Yaskawa INFORM job: DEMO_ROOF_UPPER_0625_3PAINT_21.JBI

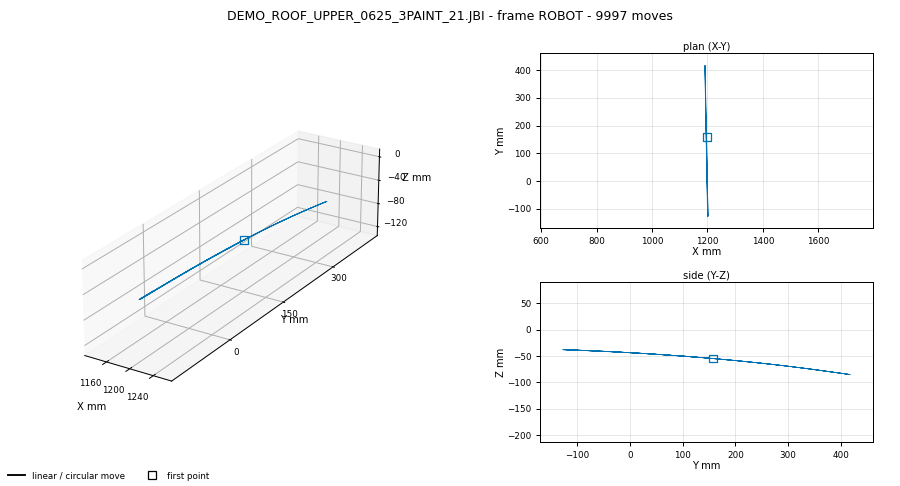
[picture p0: tool path of DEMO_ROOF_UPPER_0625_3PAINT_21.JBI in frame ROBOT, 9997 of 9997 moves have a stored position in this frame; points joined in program order, loops and branches not executed]
/JOB
//NAME DEMO_ROOF_UPPER_0625_3PAINT21
//POS
///NPOS 9997,0,0,0,0,0
///TOOL 0
///USER 0
///POSTYPE ROBOT
///RECTAN
///RCONF 1,0,0,0,0,0,0,0,0,0,0,0,0,0,0,0,0,0,0,0,0,0,0,0
C00000=1196.733,158.138,-54.632,-178.137,6.234,148.575
C00001=1196.739,157.889,-54.611,-178.140,6.232,148.575
C00002=1196.743,157.640,-54.589,-178.143,6.230,148.576
C00003=1196.748,157.391,-54.568,-178.145,6.229,148.576
C00004=1196.752,157.142,-54.547,-178.147,6.227,148.576
C00005=1196.757,156.894,-54.525,-178.150,6.226,148.577
C00006=1196.762,156.644,-54.504,-178.153,6.224,148.577
C00007=1196.766,156.395,-54.482,-178.156,6.222,148.578
C00008=1196.771,156.146,-54.460,-178.158,6.222,148.578
C00009=1196.776,155.896,-54.439,-178.161,6.220,148.579
C00010=1196.780,155.648,-54.418,-178.163,6.218,148.579
C00011=1196.785,155.399,-54.397,-178.166,6.216,148.579
C00012=1196.790,155.150,-54.375,-178.169,6.216,148.580
C00013=1196.795,154.900,-54.354,-178.171,6.214,148.580
C00014=1196.800,154.652,-54.332,-178.174,6.212,148.581
C00015=1196.804,154.403,-54.312,-178.177,6.210,148.581
C00016=1196.809,154.154,-54.290,-178.179,6.209,148.581
C00017=1196.813,153.904,-54.269,-178.182,6.208,148.582
C00018=1196.818,153.655,-54.247,-178.185,6.206,148.582
C00019=1196.823,153.406,-54.226,-178.187,6.204,148.583
C00020=1196.828,153.158,-54.205,-178.189,6.203,148.583
C00021=1196.832,152.908,-54.184,-178.192,6.201,148.584
C00022=1196.837,152.659,-54.162,-178.195,6.200,148.584
C00023=1196.841,152.410,-54.142,-178.198,6.198,148.585
C00024=1196.846,152.162,-54.120,-178.200,6.197,148.585
C00025=1196.852,151.912,-54.099,-178.203,6.196,148.585
C00026=1196.856,151.662,-54.078,-178.205,6.194,148.586
C00027=1196.860,151.414,-54.056,-178.208,6.192,148.586
C00028=1196.865,151.165,-54.036,-178.211,6.191,148.587
C00029=1196.871,150.916,-54.015,-178.213,6.190,148.587
C00030=1196.875,150.667,-53.993,-178.216,6.188,148.587
C00031=1196.880,150.418,-53.972,-178.219,6.186,148.588
C00032=1196.884,150.169,-53.950,-178.221,6.185,148.588
C00033=1196.889,149.920,-53.930,-178.224,6.184,148.589
C00034=1196.894,149.670,-53.909,-178.227,6.182,148.589
C00035=1196.899,149.421,-53.888,-178.229,6.180,148.590
C00036=1196.903,149.173,-53.867,-178.231,6.179,148.590
C00037=1196.908,148.924,-53.846,-178.235,6.178,148.591
C00038=1196.913,148.674,-53.825,-178.237,6.176,148.591
C00039=1196.917,148.425,-53.804,-178.239,6.175,148.591
C00040=1196.922,148.176,-53.783,-178.242,6.173,148.592
C00041=1196.927,147.927,-53.762,-178.245,6.171,148.592
C00042=1196.932,147.678,-53.741,-178.248,6.170,148.593
C00043=1196.937,147.429,-53.720,-178.250,6.169,148.593
C00044=1196.941,147.180,-53.699,-178.253,6.167,148.593
C00045=1196.946,146.930,-53.678,-178.255,6.165,148.594
C00046=1196.950,146.681,-53.658,-178.258,6.165,148.594
C00047=1196.955,146.432,-53.637,-178.261,6.163,148.595
C00048=1196.959,146.184,-53.616,-178.263,6.161,148.595
C00049=1196.965,145.934,-53.595,-178.266,6.159,148.596
C00050=1196.969,145.685,-53.574,-178.269,6.159,148.596
C00051=1196.974,145.436,-53.553,-178.271,6.157,148.597
C00052=1196.979,145.187,-53.533,-178.274,6.155,148.597
C00053=1196.984,144.938,-53.512,-178.276,6.154,148.597
C00054=1196.988,144.689,-53.492,-178.279,6.153,148.598
C00055=1196.993,144.440,-53.470,-178.282,6.151,148.598
C00056=1196.997,144.191,-53.449,-178.284,6.150,148.599
C00057=1197.002,143.942,-53.428,-178.287,6.148,148.599
C00058=1197.006,143.693,-53.408,-178.290,6.147,148.600
C00059=1197.012,143.443,-53.387,-178.293,6.145,148.600
C00060=1197.016,143.194,-53.366,-178.295,6.144,148.601
C00061=1197.021,142.945,-53.345,-178.297,6.142,148.601
C00062=1197.026,142.696,-53.325,-178.301,6.141,148.602
C00063=1197.031,142.447,-53.304,-178.303,6.140,148.602
C00064=1197.035,142.198,-53.284,-178.305,6.138,148.602
C00065=1197.041,141.949,-53.263,-178.308,6.137,148.603
C00066=1197.045,141.700,-53.242,-178.311,6.136,148.603
C00067=1197.049,141.451,-53.222,-178.313,6.134,148.604
C00068=1197.055,141.202,-53.201,-178.316,6.132,148.604
C00069=1197.059,140.953,-53.181,-178.318,6.131,148.604
C00070=1197.064,140.703,-53.160,-178.321,6.130,148.605
C00071=1197.069,140.454,-53.139,-178.324,6.128,148.605
C00072=1197.073,140.205,-53.119,-178.326,6.127,148.606
C00073=1197.078,139.956,-53.098,-178.329,6.126,148.606
C00074=1197.083,139.707,-53.078,-178.332,6.124,148.607
C00075=1197.087,139.458,-53.058,-178.334,6.123,148.607
C00076=1197.093,139.208,-53.037,-178.337,6.121,148.608
C00077=1197.097,138.959,-53.017,-178.340,6.120,148.608
C00078=1197.101,138.710,-52.996,-178.342,6.119,148.609
C00079=1197.107,138.461,-52.975,-178.345,6.117,148.609
C00080=1197.111,138.212,-52.955,-178.347,6.115,148.609
C00081=1197.115,137.963,-52.935,-178.350,6.115,148.610
C00082=1197.121,137.713,-52.914,-178.353,6.113,148.610
C00083=1197.125,137.465,-52.894,-178.355,6.111,148.611
C00084=1197.130,137.216,-52.874,-178.358,6.111,148.611
C00085=1197.135,136.966,-52.853,-178.361,6.109,148.612
C00086=1197.139,136.717,-52.832,-178.363,6.107,148.612
C00087=1197.144,136.468,-52.813,-178.365,6.106,148.613
C00088=1197.149,136.220,-52.793,-178.369,6.105,148.613
C00089=1197.154,135.970,-52.772,-178.371,6.103,148.614
C00090=1197.159,135.721,-52.751,-178.373,6.102,148.614
C00091=1197.164,135.472,-52.732,-178.377,6.101,148.615
C00092=1197.169,135.222,-52.711,-178.379,6.100,148.615
C00093=1197.173,134.974,-52.690,-178.381,6.098,148.615
C00094=1197.178,134.725,-52.670,-178.385,6.096,148.616
C00095=1197.182,134.475,-52.650,-178.387,6.096,148.616
C00096=1197.187,134.226,-52.630,-178.389,6.094,148.617
C00097=1197.192,133.977,-52.609,-178.393,6.092,148.617
C00098=1197.197,133.728,-52.590,-178.395,6.091,148.618
C00099=1197.202,133.479,-52.569,-178.397,6.090,148.618
C00100=1197.207,133.210,-52.548,-178.401,6.088,148.619
C00101=1197.211,132.941,-52.525,-178.403,6.087,148.619
C00102=1197.217,132.672,-52.504,-178.406,6.086,148.620
C00103=1197.222,132.404,-52.482,-178.409,6.084,148.620
C00104=1197.226,132.155,-52.462,-178.411,6.082,148.621
C00105=1197.232,131.906,-52.442,-178.414,6.082,148.621
C00106=1197.237,131.657,-52.422,-178.417,6.080,148.622
C00107=1197.241,131.408,-52.402,-178.419,6.078,148.622
C00108=1197.246,131.159,-52.381,-178.422,6.078,148.623
C00109=1197.251,130.909,-52.362,-178.425,6.076,148.623
C00110=1197.255,130.660,-52.341,-178.427,6.075,148.623
C00111=1197.260,130.411,-52.322,-178.430,6.073,148.624
C00112=1197.265,130.162,-52.302,-178.432,6.072,148.624
C00113=1197.270,129.913,-52.281,-178.435,6.071,148.625
C00114=1197.275,129.664,-52.261,-178.438,6.069,148.626
C00115=1197.279,129.414,-52.241,-178.440,6.068,148.626
C00116=1197.285,129.166,-52.221,-178.443,6.067,148.626
C00117=1197.289,128.916,-52.202,-178.446,6.065,148.627
C00118=1197.294,128.667,-52.181,-178.448,6.064,148.627
C00119=1197.298,128.418,-52.162,-178.451,6.062,148.628
C00120=1197.303,128.168,-52.142,-178.453,6.062,148.628
C00121=1197.308,127.920,-52.122,-178.456,6.060,148.629
C00122=1197.313,127.670,-52.102,-178.459,6.058,148.629
C00123=1197.317,127.421,-52.082,-178.461,6.058,148.630
C00124=1197.322,127.172,-52.062,-178.464,6.056,148.630
C00125=1197.327,126.924,-52.042,-178.466,6.055,148.631
C00126=1197.332,126.674,-52.023,-178.469,6.054,148.631
C00127=1197.337,126.424,-52.003,-178.471,6.053,148.632
C00128=1197.341,126.175,-51.983,-178.474,6.051,148.632
C00129=1197.346,125.927,-51.963,-178.477,6.049,148.633
C00130=1197.351,125.677,-51.944,-178.479,6.049,148.633
C00131=1197.356,125.428,-51.923,-178.482,6.047,148.634
C00132=1197.360,125.178,-51.904,-178.485,6.046,148.634
C00133=1197.366,124.930,-51.884,-178.487,6.044,148.634
C00134=1197.370,124.681,-51.864,-178.490,6.044,148.635
C00135=1197.375,124.431,-51.844,-178.493,6.042,148.635
C00136=1197.380,124.182,-51.825,-178.495,6.040,148.636
C00137=1197.385,123.933,-51.805,-178.498,6.040,148.636
C00138=1197.389,123.684,-51.785,-178.501,6.038,148.637
C00139=1197.394,123.434,-51.765,-178.503,6.037,148.638
C00140=1197.399,123.186,-51.747,-178.506,6.036,148.638
C00141=1197.403,122.936,-51.727,-178.508,6.035,148.638
C00142=1197.408,122.687,-51.707,-178.511,6.033,148.639
C00143=1197.413,122.438,-51.687,-178.514,6.031,148.639
C00144=1197.418,122.189,-51.668,-178.516,6.031,148.640
C00145=1197.423,121.939,-51.648,-178.519,6.029,148.640
C00146=1197.428,121.689,-51.628,-178.521,6.028,148.641
C00147=1197.433,121.441,-51.608,-178.524,6.027,148.641
C00148=1197.437,121.192,-51.589,-178.527,6.026,148.642
C00149=1197.441,120.942,-51.570,-178.529,6.024,148.642
C00150=1197.447,120.694,-51.550,-178.532,6.023,148.643
C00151=1197.451,120.444,-51.531,-178.535,6.022,148.643
C00152=1197.457,120.195,-51.511,-178.537,6.021,148.644
C00153=1197.461,119.946,-51.492,-178.540,6.019,148.644
C00154=1197.466,119.697,-51.471,-178.543,6.018,148.645
C00155=1197.471,119.448,-51.453,-178.545,6.017,148.645
C00156=1197.475,119.198,-51.433,-178.548,6.015,148.646
C00157=1197.480,118.949,-51.413,-178.550,6.014,148.646
C00158=1197.485,118.700,-51.394,-178.553,6.013,148.647
C00159=1197.489,118.451,-51.375,-178.555,6.012,148.647
C00160=1197.495,118.202,-51.356,-178.558,6.011,148.648
C00161=1197.499,117.952,-51.336,-178.561,6.010,148.648
C00162=1197.504,117.703,-51.316,-178.563,6.008,148.649
C00163=1197.510,117.454,-51.297,-178.566,6.007,148.649
C00164=1197.514,117.205,-51.278,-178.569,6.005,148.650
C00165=1197.519,116.956,-51.259,-178.571,6.005,148.650
C00166=1197.524,116.706,-51.239,-178.574,6.003,148.651
C00167=1197.528,116.457,-51.219,-178.577,6.003,148.651
C00168=1197.533,116.208,-51.201,-178.579,6.001,148.652
C00169=1197.538,115.959,-51.181,-178.581,6.000,148.652
C00170=1197.543,115.710,-51.162,-178.585,5.998,148.653
C00171=1197.547,115.460,-51.143,-178.587,5.998,148.653
C00172=1197.552,115.212,-51.123,-178.590,5.996,148.654
C00173=1197.557,114.962,-51.104,-178.592,5.995,148.654
C00174=1197.561,114.713,-51.085,-178.595,5.993,148.655
C00175=1197.567,114.463,-51.066,-178.597,5.993,148.655
C00176=1197.572,114.214,-51.046,-178.600,5.991,148.656
C00177=1197.577,113.965,-51.027,-178.603,5.990,148.656
C00178=1197.581,113.716,-51.008,-178.605,5.989,148.657
C00179=1197.586,113.467,-50.989,-178.608,5.988,148.657
C00180=1197.590,113.217,-50.970,-178.611,5.986,148.658
C00181=1197.596,112.969,-50.950,-178.613,5.985,148.658
C00182=1197.601,112.718,-50.931,-178.616,5.984,148.659
C00183=1197.605,112.470,-50.913,-178.618,5.983,148.659
C00184=1197.610,112.220,-50.893,-178.621,5.982,148.660
C00185=1197.615,111.971,-50.874,-178.623,5.981,148.660
C00186=1197.619,111.722,-50.855,-178.627,5.979,148.661
C00187=1197.625,111.473,-50.836,-178.629,5.978,148.661
C00188=1197.629,111.223,-50.817,-178.631,5.977,148.662
C00189=1197.634,110.974,-50.798,-178.634,5.976,148.662
C00190=1197.639,110.725,-50.778,-178.637,5.974,148.663
C00191=1197.644,110.476,-50.760,-178.639,5.974,148.663
C00192=1197.649,110.226,-50.741,-178.642,5.972,148.664
C00193=1197.653,109.978,-50.722,-178.645,5.971,148.664
C00194=1197.658,109.728,-50.702,-178.647,5.970,148.665
C00195=1197.663,109.479,-50.684,-178.650,5.969,148.665
C00196=1197.668,109.229,-50.665,-178.653,5.967,148.666
C00197=1197.672,108.981,-50.646,-178.655,5.966,148.666
C00198=1197.678,108.731,-50.627,-178.658,5.965,148.667
C00199=1197.682,108.482,-50.608,-178.660,5.964,148.667
C00200=1197.687,108.233,-50.589,-178.663,5.963,148.668
C00201=1197.692,107.983,-50.571,-178.665,5.962,148.668
C00202=1197.697,107.734,-50.551,-178.668,5.961,148.669
C00203=1197.701,107.485,-50.532,-178.671,5.959,148.669
C00204=1197.707,107.217,-50.512,-178.674,5.958,148.670
C00205=1197.712,106.949,-50.492,-178.676,5.957,148.670
C00206=1197.717,106.680,-50.472,-178.679,5.956,148.671
C00207=1197.722,106.412,-50.451,-178.682,5.955,148.672
C00208=1197.727,106.162,-50.432,-178.685,5.953,148.672
C00209=1197.732,105.913,-50.413,-178.687,5.953,148.673
C00210=1197.737,105.664,-50.395,-178.690,5.951,148.673
C00211=1197.742,105.414,-50.376,-178.692,5.950,148.674
C00212=1197.747,105.165,-50.358,-178.695,5.949,148.674
C00213=1197.752,104.916,-50.338,-178.698,5.948,148.675
C00214=1197.756,104.666,-50.320,-178.700,5.946,148.675
C00215=1197.761,104.418,-50.301,-178.703,5.946,148.676
C00216=1197.766,104.168,-50.283,-178.706,5.944,148.676
C00217=1197.770,103.919,-50.264,-178.708,5.943,148.677
C00218=1197.776,103.670,-50.245,-178.711,5.943,148.677
C00219=1197.780,103.420,-50.226,-178.713,5.941,148.678
C00220=1197.785,103.171,-50.208,-178.716,5.940,148.678
C00221=1197.790,102.922,-50.189,-178.719,5.938,148.679
C00222=1197.795,102.672,-50.171,-178.721,5.938,148.679
C00223=1197.800,102.423,-50.151,-178.724,5.936,148.680
C00224=1197.805,102.174,-50.133,-178.726,5.936,148.680
C00225=1197.809,101.924,-50.115,-178.729,5.935,148.681
C00226=1197.815,101.676,-50.096,-178.732,5.933,148.682
C00227=1197.820,101.426,-50.078,-178.734,5.932,148.682
C00228=1197.824,101.177,-50.059,-178.737,5.931,148.683
C00229=1197.829,100.928,-50.040,-178.739,5.930,148.683
C00230=1197.834,100.678,-50.022,-178.742,5.929,148.684
C00231=1197.838,100.429,-50.003,-178.745,5.928,148.684
C00232=1197.843,100.180,-49.985,-178.747,5.927,148.685
C00233=1197.849,99.931,-49.966,-178.750,5.925,148.685
C00234=1197.853,99.681,-49.947,-178.753,5.925,148.686
C00235=1197.858,99.432,-49.929,-178.755,5.923,148.686
C00236=1197.863,99.183,-49.911,-178.758,5.922,148.687
C00237=1197.868,98.934,-49.892,-178.760,5.922,148.687
C00238=1197.872,98.684,-49.874,-178.763,5.920,148.688
C00239=1197.877,98.435,-49.856,-178.765,5.919,148.688
C00240=1197.883,98.186,-49.837,-178.768,5.918,148.689
C00241=1197.887,97.937,-49.819,-178.771,5.917,148.689
C00242=1197.892,97.687,-49.800,-178.773,5.916,148.690
C00243=1197.897,97.438,-49.782,-178.776,5.915,148.690
C00244=1197.901,97.189,-49.764,-178.779,5.914,148.691
C00245=1197.906,96.939,-49.745,-178.781,5.912,148.691
C00246=1197.911,96.690,-49.727,-178.784,5.912,148.692
C00247=1197.916,96.441,-49.709,-178.786,5.911,148.693
C00248=1197.921,96.192,-49.691,-178.789,5.909,148.693
C00249=1197.926,95.942,-49.673,-178.791,5.908,148.694
C00250=1197.931,95.693,-49.653,-178.795,5.907,148.694
C00251=1197.935,95.444,-49.635,-178.797,5.906,148.695
C00252=1197.940,95.195,-49.617,-178.799,5.906,148.695
C00253=1197.945,94.945,-49.599,-178.802,5.904,148.696
C00254=1197.950,94.696,-49.581,-178.805,5.903,148.696
C00255=1197.955,94.446,-49.563,-178.807,5.903,148.697
C00256=1197.960,94.197,-49.544,-178.810,5.901,148.697
C00257=1197.965,93.948,-49.526,-178.813,5.900,148.698
C00258=1197.970,93.699,-49.507,-178.815,5.899,148.698
C00259=1197.974,93.449,-49.489,-178.818,5.898,148.699
C00260=1197.979,93.200,-49.471,-178.820,5.897,148.700
C00261=1197.984,92.951,-49.453,-178.823,5.896,148.700
C00262=1197.989,92.702,-49.435,-178.825,5.895,148.701
C00263=1197.994,92.453,-49.417,-178.828,5.894,148.701
C00264=1197.999,92.203,-49.399,-178.831,5.893,148.702
C00265=1198.003,91.953,-49.381,-178.833,5.892,148.702
C00266=1198.009,91.704,-49.362,-178.836,5.890,148.703
C00267=1198.013,91.455,-49.344,-178.839,5.890,148.703
C00268=1198.018,91.206,-49.326,-178.841,5.889,148.704
C00269=1198.023,90.956,-49.308,-178.844,5.887,148.704
C00270=1198.028,90.707,-49.290,-178.847,5.887,148.705
C00271=1198.033,90.458,-49.272,-178.849,5.886,148.706
C00272=1198.037,90.208,-49.254,-178.852,5.884,148.706
C00273=1198.042,89.959,-49.236,-178.854,5.884,148.707
C00274=1198.047,89.710,-49.218,-178.857,5.883,148.707
C00275=1198.052,89.461,-49.200,-178.859,5.881,148.708
C00276=1198.057,89.212,-49.182,-178.862,5.881,148.708
C00277=1198.062,88.962,-49.164,-178.864,5.880,148.709
C00278=1198.067,88.713,-49.146,-178.867,5.878,148.709
C00279=1198.072,88.463,-49.129,-178.870,5.878,148.710
C00280=1198.076,88.214,-49.111,-178.873,5.876,148.710
C00281=1198.081,87.964,-49.093,-178.875,5.876,148.711
C00282=1198.086,87.715,-49.075,-178.877,5.875,148.712
C00283=1198.091,87.466,-49.057,-178.881,5.873,148.712
C00284=1198.096,87.217,-49.039,-178.883,5.872,148.713
C00285=1198.101,86.968,-49.021,-178.885,5.872,148.713
C00286=1198.106,86.718,-49.003,-178.888,5.870,148.714
C00287=1198.111,86.469,-48.985,-178.891,5.869,148.714
C00288=1198.115,86.220,-48.968,-178.893,5.869,148.715
C00289=1198.120,85.971,-48.950,-178.896,5.867,148.715
C00290=1198.125,85.721,-48.932,-178.899,5.867,148.716
C00291=1198.130,85.472,-48.914,-178.901,5.866,148.716
C00292=1198.135,85.222,-48.897,-178.904,5.864,148.717
C00293=1198.140,84.973,-48.879,-178.906,5.863,148.718
C00294=1198.145,84.724,-48.861,-178.909,5.863,148.718
C00295=1198.149,84.474,-48.843,-178.912,5.861,148.719
C00296=1198.155,84.224,-48.825,-178.914,5.860,148.719
C00297=1198.159,83.975,-48.807,-178.917,5.860,148.720
C00298=1198.164,83.726,-48.790,-178.919,5.859,148.720
C00299=1198.169,83.477,-48.773,-178.922,5.858,148.721
C00300=1198.174,83.227,-48.755,-178.924,5.857,148.721
C00301=1198.179,82.978,-48.737,-178.927,5.856,148.722
C00302=1198.184,82.729,-48.719,-178.930,5.855,148.723
C00303=1198.189,82.479,-48.701,-178.932,5.854,148.723
C00304=1198.193,82.230,-48.684,-178.935,5.853,148.724
C00305=1198.198,81.981,-48.666,-178.938,5.852,148.724
C00306=1198.203,81.731,-48.649,-178.940,5.851,148.725
C00307=1198.208,81.482,-48.631,-178.942,5.850,148.725
C00308=1198.214,81.214,-48.613,-178.945,5.849,148.726
C00309=1198.219,80.946,-48.593,-178.948,5.848,148.727
C00310=1198.225,80.677,-48.574,-178.951,5.847,148.727
C00311=1198.229,80.409,-48.556,-178.954,5.846,148.728
C00312=1198.234,80.159,-48.538,-178.956,5.845,148.728
C00313=1198.239,79.910,-48.520,-178.959,5.844,148.729
C00314=1198.244,79.661,-48.502,-178.961,5.843,148.729
C00315=1198.249,79.411,-48.485,-178.964,5.842,148.730
C00316=1198.253,79.162,-48.468,-178.967,5.841,148.731
C00317=1198.258,78.912,-48.450,-178.969,5.840,148.731
C00318=1198.263,78.663,-48.432,-178.972,5.840,148.732
C00319=1198.268,78.415,-48.416,-178.974,5.839,148.732
C00320=1198.273,78.165,-48.398,-178.977,5.837,148.733
C00321=1198.279,77.916,-48.381,-178.980,5.837,148.734
C00322=1198.284,77.666,-48.363,-178.982,5.836,148.734
C00323=1198.288,77.417,-48.346,-178.985,5.834,148.735
C00324=1198.293,77.168,-48.328,-178.987,5.834,148.735
C00325=1198.298,76.918,-48.311,-178.990,5.833,148.736
C00326=1198.302,76.669,-48.294,-178.993,5.832,148.736
C00327=1198.308,76.419,-48.276,-178.995,5.831,148.737
C00328=1198.312,76.170,-48.258,-178.998,5.830,148.737
C00329=1198.317,75.921,-48.242,-179.000,5.829,148.738
C00330=1198.322,75.671,-48.224,-179.003,5.828,148.739
C00331=1198.328,75.422,-48.207,-179.006,5.827,148.739
C00332=1198.332,75.173,-48.190,-179.008,5.826,148.740
C00333=1198.337,74.924,-48.172,-179.011,5.826,148.740
C00334=1198.342,74.674,-48.155,-179.014,5.824,148.741
C00335=1198.347,74.424,-48.138,-179.016,5.824,148.741
C00336=1198.352,74.175,-48.120,-179.019,5.823,148.742
C00337=1198.357,73.925,-48.103,-179.021,5.822,148.742
C00338=1198.361,73.677,-48.086,-179.024,5.821,148.743
C00339=1198.367,73.427,-48.069,-179.027,5.820,148.744
C00340=1198.371,73.178,-48.052,-179.029,5.819,148.744
C00341=1198.376,72.929,-48.034,-179.032,5.819,148.745
C00342=1198.381,72.679,-48.017,-179.034,5.817,148.745
C00343=1198.386,72.429,-48.000,-179.037,5.816,148.746
C00344=1198.391,72.180,-47.983,-179.039,5.816,148.747
C00345=1198.396,71.932,-47.966,-179.042,5.815,148.747
C00346=1198.401,71.682,-47.949,-179.045,5.814,148.748
C00347=1198.406,71.432,-47.932,-179.047,5.813,148.748
C00348=1198.411,71.183,-47.914,-179.050,5.812,148.749
C00349=1198.415,70.934,-47.897,-179.052,5.812,148.749
C00350=1198.420,70.684,-47.880,-179.055,5.810,148.750
C00351=1198.425,70.435,-47.864,-179.058,5.809,148.751
C00352=1198.430,70.186,-47.846,-179.060,5.809,148.751
C00353=1198.435,69.936,-47.828,-179.062,5.808,148.752
C00354=1198.440,69.687,-47.812,-179.066,5.807,148.752
C00355=1198.446,69.437,-47.795,-179.068,5.806,148.753
C00356=1198.450,69.188,-47.778,-179.070,5.805,148.753
C00357=1198.454,68.939,-47.761,-179.073,5.805,148.754
C00358=1198.460,68.689,-47.744,-179.076,5.803,148.755
C00359=1198.464,68.440,-47.727,-179.078,5.802,148.755
C00360=1198.470,68.191,-47.710,-179.081,5.802,148.756
C00361=1198.474,67.941,-47.693,-179.083,5.801,148.756
C00362=1198.480,67.691,-47.676,-179.086,5.800,148.757
C00363=1198.484,67.442,-47.659,-179.089,5.799,148.758
C00364=1198.490,67.194,-47.642,-179.091,5.798,148.758
C00365=1198.494,66.944,-47.625,-179.094,5.797,148.759
C00366=1198.499,66.694,-47.608,-179.096,5.797,148.759
C00367=1198.504,66.445,-47.591,-179.099,5.795,148.760
C00368=1198.509,66.196,-47.575,-179.102,5.795,148.760
C00369=1198.514,65.946,-47.558,-179.104,5.794,148.761
C00370=1198.519,65.697,-47.541,-179.106,5.793,148.761
C00371=1198.524,65.447,-47.524,-179.109,5.793,148.762
C00372=1198.529,65.198,-47.507,-179.112,5.791,148.763
C00373=1198.533,64.949,-47.491,-179.114,5.790,148.763
C00374=1198.539,64.699,-47.473,-179.117,5.790,148.764
C00375=1198.543,64.449,-47.457,-179.120,5.789,148.765
C00376=1198.548,64.201,-47.441,-179.122,5.788,148.765
C00377=1198.553,63.951,-47.423,-179.125,5.787,148.766
C00378=1198.558,63.701,-47.407,-179.128,5.786,148.766
C00379=1198.564,63.452,-47.390,-179.130,5.786,148.767
C00380=1198.568,63.203,-47.373,-179.132,5.785,148.767
C00381=1198.573,62.953,-47.356,-179.135,5.784,148.768
C00382=1198.578,62.704,-47.339,-179.138,5.783,148.768
C00383=1198.583,62.455,-47.323,-179.140,5.782,148.769
C00384=1198.587,62.205,-47.306,-179.143,5.781,148.770
C00385=1198.593,61.956,-47.289,-179.145,5.781,148.770
C00386=1198.598,61.707,-47.273,-179.148,5.780,148.771
C00387=1198.602,61.457,-47.256,-179.151,5.778,148.771
C00388=1198.607,61.208,-47.240,-179.153,5.778,148.772
C00389=1198.613,60.958,-47.223,-179.156,5.777,148.773
C00390=1198.617,60.708,-47.206,-179.158,5.776,148.773
C00391=1198.622,60.460,-47.190,-179.161,5.776,148.774
C00392=1198.628,60.210,-47.173,-179.164,5.775,148.774
C00393=1198.632,59.960,-47.156,-179.166,5.774,148.775
C00394=1198.637,59.712,-47.140,-179.169,5.773,148.776
C00395=1198.642,59.462,-47.123,-179.171,5.773,148.776
C00396=1198.648,59.212,-47.107,-179.174,5.772,148.777
C00397=1198.652,58.963,-47.090,-179.176,5.771,148.777
C00398=1198.657,58.713,-47.074,-179.179,5.770,148.778
C00399=1198.662,58.465,-47.057,-179.182,5.769,148.779
C00400=1198.666,58.215,-47.041,-179.184,5.768,148.779
C00401=1198.672,57.965,-47.024,-179.187,5.768,148.780
C00402=1198.677,57.716,-47.008,-179.189,5.767,148.780
C00403=1198.681,57.466,-46.991,-179.191,5.766,148.781
C00404=1198.686,57.218,-46.975,-179.195,5.765,148.781
C00405=1198.692,56.968,-46.958,-179.197,5.764,148.782
C00406=1198.697,56.718,-46.942,-179.199,5.764,148.783
C00407=1198.702,56.469,-46.925,-179.202,5.763,148.783
C00408=1198.706,56.220,-46.909,-179.205,5.763,148.784
C00409=1198.711,55.970,-46.893,-179.207,5.762,148.784
C00410=1198.716,55.721,-46.876,-179.210,5.760,148.785
C00411=1198.722,55.472,-46.859,-179.213,5.760,148.786
C00412=1198.727,55.202,-46.842,-179.215,5.759,148.786
C00413=1198.732,54.934,-46.824,-179.218,5.759,148.787
C00414=1198.737,54.666,-46.807,-179.221,5.757,148.787
C00415=1198.742,54.397,-46.789,-179.223,5.756,148.788
C00416=1198.747,54.148,-46.774,-179.226,5.756,148.789
C00417=1198.753,53.898,-46.756,-179.229,5.755,148.789
C00418=1198.758,53.649,-46.740,-179.231,5.754,148.790
C00419=1198.763,53.399,-46.724,-179.234,5.753,148.791
C00420=1198.768,53.151,-46.708,-179.237,5.753,148.791
C00421=1198.772,52.900,-46.692,-179.239,5.752,148.792
C00422=1198.778,52.652,-46.676,-179.241,5.751,148.792
C00423=1198.782,52.402,-46.659,-179.244,5.751,148.793
C00424=1198.787,52.153,-46.643,-179.247,5.750,148.794
C00425=1198.792,51.903,-46.627,-179.249,5.749,148.794
C00426=1198.797,51.654,-46.611,-179.252,5.748,148.795
C00427=1198.802,51.404,-46.594,-179.255,5.747,148.795
C00428=1198.807,51.155,-46.579,-179.257,5.746,148.796
C00429=1198.812,50.906,-46.562,-179.259,5.746,148.797
C00430=1198.817,50.657,-46.546,-179.262,5.745,148.797
C00431=1198.821,50.407,-46.530,-179.265,5.745,148.798
C00432=1198.827,50.158,-46.514,-179.267,5.744,148.798
C00433=1198.831,49.908,-46.498,-179.270,5.743,148.799
C00434=1198.837,49.659,-46.481,-179.273,5.742,148.800
C00435=1198.842,49.409,-46.465,-179.275,5.741,148.800
C00436=1198.846,49.160,-46.449,-179.278,5.741,148.801
C00437=1198.851,48.910,-46.433,-179.280,5.740,148.801
C00438=1198.856,48.661,-46.418,-179.283,5.739,148.802
C00439=1198.861,48.411,-46.401,-179.285,5.739,148.803
C00440=1198.866,48.162,-46.385,-179.288,5.738,148.803
C00441=1198.871,47.912,-46.369,-179.290,5.738,148.804
C00442=1198.876,47.663,-46.353,-179.293,5.736,148.804
C00443=1198.881,47.414,-46.337,-179.296,5.735,148.805
C00444=1198.886,47.164,-46.321,-179.298,5.735,148.806
C00445=1198.891,46.915,-46.305,-179.301,5.734,148.806
C00446=1198.896,46.665,-46.288,-179.303,5.733,148.807
C00447=1198.901,46.416,-46.273,-179.306,5.733,148.807
C00448=1198.906,46.166,-46.256,-179.308,5.732,148.808
C00449=1198.911,45.917,-46.241,-179.310,5.731,148.809
C00450=1198.917,45.667,-46.225,-179.313,5.731,148.809
C00451=1198.921,45.418,-46.208,-179.316,5.730,148.810
C00452=1198.926,45.168,-46.193,-179.319,5.729,148.811
C00453=1198.930,44.919,-46.177,-179.321,5.728,148.811
C00454=1198.936,44.670,-46.161,-179.324,5.728,148.812
C00455=1198.941,44.421,-46.146,-179.326,5.727,148.812
C00456=1198.946,44.170,-46.130,-179.329,5.726,148.813
C00457=1198.951,43.921,-46.114,-179.331,5.726,148.813
C00458=1198.956,43.672,-46.098,-179.334,5.725,148.814
C00459=1198.961,43.422,-46.082,-179.336,5.725,148.815
C00460=1198.966,43.173,-46.066,-179.339,5.724,148.815
C00461=1198.970,42.924,-46.050,-179.341,5.723,148.816
C00462=1198.975,42.674,-46.034,-179.344,5.722,148.817
C00463=1198.981,42.425,-46.019,-179.347,5.721,148.817
C00464=1198.986,42.175,-46.003,-179.349,5.720,148.818
C00465=1198.991,41.925,-45.987,-179.352,5.720,148.818
C00466=1198.996,41.676,-45.971,-179.355,5.719,148.819
C00467=1199.000,41.427,-45.956,-179.357,5.718,148.820
C00468=1199.006,41.177,-45.940,-179.359,5.718,148.820
C00469=1199.011,40.928,-45.925,-179.362,5.717,148.821
C00470=1199.016,40.678,-45.909,-179.365,5.717,148.822
C00471=1199.021,40.429,-45.892,-179.367,5.716,148.822
C00472=1199.025,40.180,-45.877,-179.369,5.715,148.823
C00473=1199.030,39.930,-45.861,-179.372,5.715,148.823
C00474=1199.036,39.680,-45.846,-179.375,5.714,148.824
C00475=1199.041,39.431,-45.830,-179.377,5.713,148.824
C00476=1199.046,39.182,-45.815,-179.380,5.712,148.825
C00477=1199.050,38.932,-45.799,-179.383,5.712,148.826
C00478=1199.056,38.683,-45.783,-179.385,5.711,148.826
C00479=1199.061,38.434,-45.767,-179.387,5.710,148.827
C00480=1199.065,38.184,-45.752,-179.390,5.710,148.828
C00481=1199.070,37.934,-45.736,-179.393,5.709,148.828
C00482=1199.076,37.685,-45.721,-179.395,5.709,148.829
C00483=1199.081,37.436,-45.705,-179.398,5.708,148.829
C00484=1199.085,37.186,-45.690,-179.400,5.707,148.830
C00485=1199.091,36.936,-45.674,-179.403,5.707,148.831
C00486=1199.096,36.687,-45.659,-179.405,5.706,148.831
C00487=1199.101,36.438,-45.644,-179.408,5.705,148.832
C00488=1199.105,36.188,-45.628,-179.410,5.705,148.833
C00489=1199.111,35.938,-45.612,-179.413,5.704,148.833
C00490=1199.115,35.689,-45.597,-179.416,5.704,148.834
C00491=1199.121,35.440,-45.582,-179.418,5.702,148.834
C00492=1199.126,35.190,-45.566,-179.421,5.702,148.835
C00493=1199.130,34.941,-45.551,-179.424,5.701,148.836
C00494=1199.136,34.691,-45.535,-179.426,5.700,148.836
C00495=1199.141,34.442,-45.519,-179.428,5.700,148.837
C00496=1199.145,34.192,-45.504,-179.431,5.699,148.837
C00497=1199.150,33.943,-45.488,-179.434,5.699,148.838
C00498=1199.156,33.693,-45.473,-179.436,5.698,148.839
C00499=1199.160,33.444,-45.458,-179.438,5.697,148.839
C00500=1199.165,33.194,-45.442,-179.441,5.697,148.840
C00501=1199.170,32.945,-45.427,-179.444,5.696,148.841
C00502=1199.175,32.696,-45.411,-179.446,5.696,148.841
C00503=1199.181,32.446,-45.396,-179.449,5.695,148.842
C00504=1199.186,32.196,-45.381,-179.451,5.694,148.842
C00505=1199.190,31.946,-45.366,-179.454,5.694,148.843
C00506=1199.195,31.697,-45.351,-179.456,5.693,148.844
C00507=1199.200,31.448,-45.335,-179.459,5.692,148.844
C00508=1199.205,31.199,-45.320,-179.461,5.692,148.845
C00509=1199.211,30.949,-45.304,-179.464,5.691,148.846
C00510=1199.216,30.700,-45.289,-179.467,5.691,148.846
C00511=1199.220,30.450,-45.274,-179.469,5.690,148.847
C00512=1199.226,30.200,-45.259,-179.471,5.689,148.847
C00513=1199.230,29.951,-45.244,-179.474,5.689,148.848
C00514=1199.236,29.702,-45.228,-179.477,5.688,148.849
C00515=1199.240,29.453,-45.213,-179.479,5.688,148.849
C00516=1199.246,29.183,-45.197,-179.483,5.686,148.850
C00517=1199.251,28.915,-45.181,-179.485,5.686,148.851
C00518=1199.257,28.646,-45.164,-179.488,5.685,148.851
C00519=1199.263,28.377,-45.148,-179.490,5.685,148.852
C00520=1199.267,28.128,-45.133,-179.493,5.684,148.853
C00521=1199.272,27.878,-45.117,-179.495,5.684,148.853
C00522=1199.277,27.628,-45.102,-179.498,5.683,148.854
C00523=1199.282,27.379,-45.087,-179.501,5.682,148.855
C00524=1199.287,27.130,-45.072,-179.503,5.682,148.855
C00525=1199.292,26.881,-45.057,-179.505,5.681,148.856
C00526=1199.298,26.631,-45.042,-179.508,5.681,148.856
C00527=1199.302,26.382,-45.027,-179.511,5.680,148.857
C00528=1199.308,26.132,-45.011,-179.513,5.679,148.858
C00529=1199.312,25.882,-44.997,-179.515,5.679,148.858
C00530=1199.317,25.632,-44.981,-179.518,5.678,148.859
C00531=1199.322,25.383,-44.966,-179.521,5.678,148.860
C00532=1199.327,25.133,-44.952,-179.523,5.677,148.860
C00533=1199.332,24.884,-44.936,-179.526,5.676,148.861
C00534=1199.337,24.635,-44.921,-179.528,5.676,148.861
C00535=1199.343,24.385,-44.906,-179.531,5.675,148.862
C00536=1199.347,24.136,-44.891,-179.533,5.675,148.863
C00537=1199.352,23.886,-44.877,-179.536,5.674,148.863
C00538=1199.358,23.637,-44.862,-179.538,5.673,148.864
C00539=1199.362,23.388,-44.847,-179.541,5.673,148.865
C00540=1199.368,23.138,-44.832,-179.544,5.672,148.865
C00541=1199.373,22.889,-44.817,-179.546,5.672,148.866
C00542=1199.378,22.639,-44.802,-179.548,5.671,148.866
C00543=1199.383,22.389,-44.787,-179.551,5.670,148.867
C00544=1199.388,22.140,-44.773,-179.554,5.670,148.868
C00545=1199.393,21.891,-44.758,-179.556,5.669,148.868
C00546=1199.397,21.641,-44.742,-179.559,5.669,148.869
C00547=1199.402,21.391,-44.727,-179.561,5.668,148.870
C00548=1199.407,21.142,-44.712,-179.564,5.667,148.870
C00549=1199.413,20.892,-44.698,-179.566,5.667,148.871
C00550=1199.417,20.643,-44.683,-179.569,5.666,148.872
C00551=1199.422,20.393,-44.668,-179.571,5.666,148.872
C00552=1199.428,20.144,-44.653,-179.574,5.665,148.873
C00553=1199.433,19.894,-44.638,-179.577,5.665,148.873
C00554=1199.438,19.644,-44.624,-179.579,5.664,148.874
C00555=1199.443,19.395,-44.609,-179.582,5.664,148.875
C00556=1199.448,19.145,-44.594,-179.584,5.663,148.875
C00557=1199.453,18.896,-44.579,-179.587,5.662,148.876
C00558=1199.457,18.646,-44.565,-179.589,5.662,148.877
C00559=1199.463,18.397,-44.549,-179.592,5.661,148.877
C00560=1199.468,18.147,-44.535,-179.595,5.661,148.878
C00561=1199.473,17.898,-44.521,-179.597,5.660,148.878
C00562=1199.478,17.649,-44.506,-179.599,5.660,148.879
C00563=1199.484,17.399,-44.491,-179.601,5.660,148.880
C00564=1199.488,17.150,-44.476,-179.604,5.659,148.880
C00565=1199.493,16.900,-44.462,-179.607,5.659,148.881
C00566=1199.498,16.650,-44.448,-179.609,5.658,148.882
C00567=1199.503,16.401,-44.433,-179.612,5.657,148.882
C00568=1199.509,16.151,-44.418,-179.614,5.657,148.883
C00569=1199.514,15.902,-44.404,-179.617,5.656,148.884
C00570=1199.518,15.653,-44.389,-179.620,5.656,148.884
C00571=1199.523,15.403,-44.374,-179.622,5.655,148.885
C00572=1199.528,15.153,-44.360,-179.624,5.654,148.885
C00573=1199.534,14.904,-44.344,-179.627,5.654,148.886
C00574=1199.538,14.654,-44.330,-179.630,5.653,148.887
C00575=1199.543,14.404,-44.316,-179.632,5.653,148.888
C00576=1199.548,14.155,-44.301,-179.634,5.652,148.888
C00577=1199.553,13.905,-44.287,-179.637,5.651,148.889
C00578=1199.559,13.656,-44.273,-179.640,5.651,148.889
C00579=1199.564,13.406,-44.258,-179.642,5.650,148.890
C00580=1199.569,13.157,-44.243,-179.645,5.650,148.891
C00581=1199.574,12.908,-44.229,-179.647,5.650,148.891
C00582=1199.579,12.658,-44.214,-179.649,5.649,148.892
C00583=1199.584,12.408,-44.200,-179.652,5.649,148.893
C00584=1199.588,12.159,-44.185,-179.655,5.648,148.893
C00585=1199.593,11.909,-44.171,-179.657,5.648,148.894
C00586=1199.598,11.660,-44.157,-179.659,5.647,148.894
C00587=1199.605,11.410,-44.142,-179.662,5.646,148.895
C00588=1199.610,11.161,-44.128,-179.665,5.646,148.896
C00589=1199.614,10.912,-44.113,-179.667,5.645,148.896
C00590=1199.619,10.662,-44.098,-179.670,5.645,148.897
C00591=1199.624,10.412,-44.084,-179.672,5.644,148.898
C00592=1199.629,10.162,-44.070,-179.675,5.644,148.898
C00593=1199.634,9.913,-44.056,-179.677,5.643,148.899
C00594=1199.640,9.664,-44.042,-179.680,5.643,148.900
C00595=1199.645,9.414,-44.027,-179.683,5.642,148.900
C00596=1199.649,9.165,-44.012,-179.684,5.642,148.901
C00597=1199.654,8.915,-43.998,-179.687,5.642,148.901
C00598=1199.659,8.666,-43.984,-179.690,5.641,148.902
C00599=1199.664,8.416,-43.970,-179.692,5.641,148.903
C00600=1199.670,8.167,-43.956,-179.695,5.640,148.903
C00601=1199.675,7.917,-43.941,-179.697,5.639,148.904
C00602=1199.680,7.667,-43.927,-179.700,5.639,148.905
C00603=1199.685,7.418,-43.913,-179.702,5.638,148.905
C00604=1199.689,7.168,-43.899,-179.705,5.638,148.906
C00605=1199.695,6.919,-43.885,-179.708,5.637,148.907
C00606=1199.700,6.669,-43.870,-179.710,5.637,148.907
C00607=1199.705,6.420,-43.856,-179.712,5.637,148.908
C00608=1199.710,6.170,-43.842,-179.715,5.636,148.909
C00609=1199.715,5.920,-43.828,-179.717,5.636,148.909
C00610=1199.720,5.671,-43.814,-179.720,5.635,148.910
C00611=1199.725,5.421,-43.799,-179.723,5.635,148.911
C00612=1199.730,5.172,-43.785,-179.725,5.634,148.911
C00613=1199.735,4.922,-43.771,-179.727,5.633,148.912
C00614=1199.740,4.672,-43.757,-179.730,5.633,148.912
C00615=1199.746,4.423,-43.743,-179.733,5.632,148.913
C00616=1199.751,4.174,-43.728,-179.735,5.632,148.914
C00617=1199.756,3.924,-43.714,-179.737,5.632,148.914
C00618=1199.761,3.674,-43.700,-179.740,5.631,148.915
C00619=1199.766,3.425,-43.686,-179.742,5.631,148.916
C00620=1199.772,3.156,-43.671,-179.745,5.630,148.916
C00621=1199.777,2.887,-43.655,-179.747,5.630,148.917
C00622=1199.782,2.617,-43.640,-179.750,5.629,148.918
C00623=1199.788,2.348,-43.625,-179.753,5.629,148.918
C00624=1199.793,2.099,-43.611,-179.755,5.628,148.919
C00625=1199.798,1.849,-43.597,-179.758,5.628,148.920
C00626=1199.802,1.600,-43.583,-179.761,5.627,148.920
C00627=1199.807,1.350,-43.569,-179.763,5.627,148.921
C00628=1199.813,1.101,-43.555,-179.766,5.626,148.922
C00629=1199.818,0.852,-43.541,-179.768,5.625,148.922
C00630=1199.823,0.601,-43.527,-179.771,5.625,148.923
C00631=1199.829,0.352,-43.513,-179.773,5.625,148.924
C00632=1199.834,0.102,-43.499,-179.776,5.625,148.924
C00633=1199.838,-0.147,-43.485,-179.778,5.624,148.925
C00634=1199.843,-0.396,-43.472,-179.780,5.623,148.925
C00635=1199.848,-0.646,-43.457,-179.783,5.623,148.926
C00636=1199.854,-0.896,-43.444,-179.786,5.622,148.927
C00637=1199.859,-1.145,-43.430,-179.788,5.622,148.928
C00638=1199.863,-1.394,-43.416,-179.791,5.621,148.928
C00639=1199.868,-1.644,-43.402,-179.793,5.621,148.929
C00640=1199.874,-1.894,-43.388,-179.795,5.621,148.929
C00641=1199.879,-2.143,-43.374,-179.798,5.620,148.930
C00642=1199.884,-2.393,-43.360,-179.801,5.620,148.931
C00643=1199.888,-2.643,-43.346,-179.803,5.619,148.931
C00644=1199.894,-2.892,-43.333,-179.806,5.619,148.932
C00645=1199.899,-3.142,-43.319,-179.808,5.618,148.933
C00646=1199.905,-3.391,-43.305,-179.811,5.618,148.933
C00647=1199.909,-3.640,-43.291,-179.813,5.618,148.934
C00648=1199.914,-3.891,-43.278,-179.815,5.617,148.935
C00649=1199.920,-4.140,-43.264,-179.818,5.617,148.935
C00650=1199.925,-4.389,-43.250,-179.821,5.616,148.936
C00651=1199.929,-4.639,-43.237,-179.823,5.616,148.937
C00652=1199.935,-4.888,-43.223,-179.826,5.615,148.937
C00653=1199.940,-5.138,-43.208,-179.828,5.615,148.938
C00654=1199.945,-5.388,-43.195,-179.830,5.615,148.939
C00655=1199.950,-5.637,-43.182,-179.833,5.614,148.939
C00656=1199.955,-5.887,-43.167,-179.836,5.614,148.940
C00657=1199.961,-6.136,-43.154,-179.838,5.613,148.940
C00658=1199.965,-6.386,-43.140,-179.840,5.613,148.941
C00659=1199.970,-6.636,-43.127,-179.843,5.612,148.942
C00660=1199.976,-6.885,-43.113,-179.846,5.612,148.943
C00661=1199.980,-7.135,-43.099,-179.848,5.612,148.943
C00662=1199.986,-7.384,-43.086,-179.850,5.611,148.944
C00663=1199.991,-7.634,-43.072,-179.853,5.611,148.944
C00664=1199.995,-7.884,-43.059,-179.855,5.610,148.945
C00665=1200.001,-8.133,-43.045,-179.858,5.610,148.946
C00666=1200.006,-8.383,-43.031,-179.861,5.609,148.946
C00667=1200.011,-8.632,-43.018,-179.863,5.609,148.947
C00668=1200.016,-8.882,-43.004,-179.865,5.609,148.948
C00669=1200.022,-9.131,-42.991,-179.868,5.608,148.948
C00670=1200.026,-9.381,-42.977,-179.870,5.608,148.949
C00671=1200.031,-9.631,-42.963,-179.873,5.607,148.950
C00672=1200.036,-9.880,-42.950,-179.875,5.607,148.950
C00673=1200.041,-10.130,-42.936,-179.878,5.607,148.951
C00674=1200.047,-10.379,-42.923,-179.880,5.607,148.952
C00675=1200.051,-10.629,-42.910,-179.882,5.606,148.952
C00676=1200.057,-10.878,-42.896,-179.885,5.605,148.953
C00677=1200.061,-11.128,-42.883,-179.888,5.605,148.954
C00678=1200.067,-11.377,-42.869,-179.890,5.604,148.954
C00679=1200.072,-11.627,-42.855,-179.892,5.605,148.955
C00680=1200.077,-11.877,-42.843,-179.895,5.604,148.956
C00681=1200.082,-12.126,-42.828,-179.897,5.603,148.956
C00682=1200.087,-12.376,-42.816,-179.900,5.603,148.957
C00683=1200.092,-12.626,-42.801,-179.903,5.602,148.957
C00684=1200.097,-12.875,-42.789,-179.905,5.602,148.958
C00685=1200.102,-13.125,-42.775,-179.907,5.602,148.959
C00686=1200.107,-13.374,-42.762,-179.910,5.602,148.960
C00687=1200.113,-13.624,-42.748,-179.912,5.601,148.960
C00688=1200.118,-13.873,-42.734,-179.915,5.600,148.961
C00689=1200.123,-14.123,-42.722,-179.917,5.600,148.961
C00690=1200.129,-14.373,-42.708,-179.920,5.600,148.962
C00691=1200.133,-14.622,-42.695,-179.922,5.600,148.963
C00692=1200.139,-14.872,-42.681,-179.925,5.599,148.964
C00693=1200.143,-15.121,-42.668,-179.927,5.598,148.964
C00694=1200.149,-15.371,-42.655,-179.930,5.598,148.965
C00695=1200.153,-15.621,-42.642,-179.932,5.598,148.965
C00696=1200.159,-15.870,-42.628,-179.934,5.598,148.966
C00697=1200.163,-16.120,-42.615,-179.937,5.597,148.967
C00698=1200.169,-16.370,-42.602,-179.940,5.597,148.967
C00699=1200.174,-16.620,-42.589,-179.942,5.596,148.968
C00700=1200.179,-16.868,-42.575,-179.945,5.595,148.969
C00701=1200.184,-17.119,-42.562,-179.947,5.596,148.969
C00702=1200.189,-17.368,-42.549,-179.949,5.595,148.970
C00703=1200.195,-17.617,-42.535,-179.952,5.595,148.971
C00704=1200.199,-17.867,-42.522,-179.955,5.594,148.971
C00705=1200.205,-18.117,-42.509,-179.957,5.593,148.972
C00706=1200.210,-18.367,-42.496,-179.959,5.594,148.973
C00707=1200.215,-18.616,-42.482,-179.961,5.593,148.973
C00708=1200.220,-18.866,-42.469,-179.964,5.593,148.974
C00709=1200.225,-19.115,-42.457,-179.967,5.592,148.975
C00710=1200.231,-19.365,-42.443,-179.969,5.593,148.975
C00711=1200.235,-19.615,-42.430,-179.972,5.592,148.976
C00712=1200.241,-19.864,-42.416,-179.974,5.591,148.976
C00713=1200.245,-20.114,-42.404,-179.976,5.591,148.977
C00714=1200.250,-20.363,-42.391,-179.979,5.590,148.978
C00715=1200.256,-20.613,-42.378,-179.981,5.591,148.979
C00716=1200.261,-20.863,-42.365,-179.984,5.590,148.979
C00717=1200.266,-21.112,-42.352,-179.986,5.590,148.980
C00718=1200.271,-21.361,-42.338,-179.989,5.589,148.980
C00719=1200.276,-21.611,-42.325,-179.991,5.588,148.981
C00720=1200.282,-21.861,-42.312,-179.993,5.589,148.982
C00721=1200.286,-22.111,-42.299,-179.996,5.588,148.983
C00722=1200.291,-22.360,-42.287,-179.999,5.588,148.983
C00723=1200.297,-22.610,-42.273,179.999,5.587,148.984
C00724=1200.302,-22.879,-42.260,179.996,5.587,148.985
C00725=1200.308,-23.149,-42.245,179.993,5.586,148.985
C00726=1200.313,-23.418,-42.231,179.991,5.587,148.986
C00727=1200.319,-23.688,-42.217,179.989,5.586,148.987
C00728=1200.324,-23.937,-42.204,179.986,5.586,148.987
C00729=1200.329,-24.187,-42.191,179.983,5.585,148.988
C00730=1200.335,-24.437,-42.178,179.981,5.584,148.989
C00731=1200.340,-24.686,-42.166,179.979,5.585,148.989
C00732=1200.344,-24.936,-42.153,179.976,5.584,148.990
C00733=1200.349,-25.185,-42.140,179.974,5.584,148.991
C00734=1200.355,-25.435,-42.127,179.971,5.583,148.991
C00735=1200.360,-25.685,-42.114,179.968,5.583,148.992
C00736=1200.365,-25.934,-42.101,179.967,5.583,148.992
C00737=1200.370,-26.184,-42.089,179.964,5.582,148.993
C00738=1200.375,-26.434,-42.075,179.961,5.582,148.994
C00739=1200.380,-26.683,-42.063,179.959,5.581,148.995
C00740=1200.385,-26.933,-42.050,179.957,5.582,148.995
C00741=1200.390,-27.183,-42.037,179.954,5.581,148.996
C00742=1200.396,-27.432,-42.024,179.952,5.581,148.996
C00743=1200.401,-27.682,-42.011,179.949,5.580,148.997
C00744=1200.405,-27.932,-41.998,179.947,5.580,148.998
C00745=1200.411,-28.181,-41.986,179.945,5.580,148.999
C00746=1200.416,-28.430,-41.973,179.942,5.579,148.999
C00747=1200.422,-28.680,-41.960,179.939,5.579,149.000
C00748=1200.426,-28.930,-41.947,179.937,5.579,149.001
C00749=1200.431,-29.179,-41.934,179.935,5.578,149.001
C00750=1200.436,-29.429,-41.922,179.932,5.578,149.002
C00751=1200.441,-29.678,-41.909,179.930,5.578,149.002
C00752=1200.447,-29.929,-41.896,179.928,5.578,149.003
C00753=1200.452,-30.178,-41.884,179.925,5.577,149.004
C00754=1200.457,-30.427,-41.871,179.922,5.577,149.005
C00755=1200.462,-30.677,-41.858,179.920,5.576,149.005
C00756=1200.467,-30.927,-41.845,179.918,5.576,149.006
C00757=1200.472,-31.176,-41.833,179.915,5.576,149.006
C00758=1200.478,-31.426,-41.820,179.913,5.575,149.007
C00759=1200.483,-31.676,-41.808,179.910,5.575,149.008
C00760=1200.488,-31.926,-41.795,179.908,5.575,149.009
C00761=1200.493,-32.175,-41.782,179.906,5.575,149.009
C00762=1200.498,-32.424,-41.770,179.903,5.574,149.010
C00763=1200.503,-32.674,-41.757,179.900,5.574,149.010
C00764=1200.508,-32.924,-41.744,179.898,5.574,149.011
C00765=1200.513,-33.174,-41.732,179.896,5.573,149.012
C00766=1200.518,-33.423,-41.720,179.893,5.573,149.013
C00767=1200.524,-33.673,-41.706,179.891,5.572,149.013
C00768=1200.529,-33.922,-41.694,179.889,5.573,149.014
C00769=1200.534,-34.172,-41.682,179.886,5.572,149.014
C00770=1200.539,-34.422,-41.669,179.883,5.572,149.015
C00771=1200.544,-34.671,-41.656,179.881,5.571,149.016
C00772=1200.550,-34.920,-41.644,179.879,5.571,149.016
C00773=1200.555,-35.170,-41.632,179.876,5.571,149.017
C00774=1200.559,-35.420,-41.619,179.874,5.570,149.018
C00775=1200.565,-35.670,-41.606,179.872,5.570,149.018
C00776=1200.570,-35.919,-41.594,179.869,5.570,149.019
C00777=1200.575,-36.169,-41.582,179.866,5.570,149.020
C00778=1200.580,-36.418,-41.569,179.864,5.569,149.020
C00779=1200.585,-36.668,-41.557,179.862,5.569,149.021
C00780=1200.590,-36.918,-41.544,179.860,5.569,149.022
C00781=1200.595,-37.168,-41.532,179.857,5.568,149.022
C00782=1200.600,-37.417,-41.519,179.854,5.568,149.023
C00783=1200.606,-37.667,-41.507,179.852,5.568,149.024
C00784=1200.611,-37.916,-41.495,179.849,5.568,149.024
C00785=1200.616,-38.165,-41.482,179.847,5.567,149.025
C00786=1200.622,-38.415,-41.470,179.845,5.567,149.026
C00787=1200.627,-38.665,-41.458,179.843,5.567,149.026
C00788=1200.632,-38.915,-41.445,179.840,5.566,149.027
C00789=1200.637,-39.165,-41.433,179.837,5.566,149.028
C00790=1200.642,-39.414,-41.420,179.835,5.566,149.028
C00791=1200.647,-39.664,-41.408,179.832,5.566,149.029
C00792=1200.652,-39.913,-41.396,179.830,5.565,149.030
C00793=1200.658,-40.163,-41.384,179.828,5.565,149.030
C00794=1200.663,-40.412,-41.371,179.826,5.565,149.031
C00795=1200.668,-40.662,-41.359,179.823,5.564,149.032
C00796=1200.673,-40.912,-41.346,179.820,5.564,149.032
C00797=1200.678,-41.162,-41.334,179.818,5.564,149.033
C00798=1200.683,-41.412,-41.322,179.816,5.563,149.034
C00799=1200.689,-41.661,-41.309,179.813,5.563,149.034
C00800=1200.694,-41.911,-41.297,179.811,5.563,149.035
C00801=1200.699,-42.160,-41.285,179.809,5.563,149.036
C00802=1200.704,-42.410,-41.273,179.806,5.562,149.036
C00803=1200.709,-42.659,-41.261,179.804,5.563,149.037
C00804=1200.714,-42.909,-41.249,179.801,5.562,149.038
C00805=1200.719,-43.158,-41.236,179.799,5.561,149.038
C00806=1200.725,-43.408,-41.224,179.796,5.561,149.039
C00807=1200.730,-43.658,-41.212,179.794,5.561,149.040
C00808=1200.735,-43.908,-41.200,179.792,5.561,149.040
C00809=1200.740,-44.158,-41.187,179.789,5.560,149.041
C00810=1200.745,-44.408,-41.175,179.787,5.561,149.042
C00811=1200.750,-44.657,-41.163,179.785,5.560,149.042
C00812=1200.755,-44.907,-41.151,179.782,5.559,149.043
C00813=1200.761,-45.156,-41.139,179.780,5.560,149.044
C00814=1200.766,-45.406,-41.127,179.777,5.559,149.044
C00815=1200.771,-45.656,-41.115,179.775,5.559,149.045
C00816=1200.776,-45.905,-41.102,179.773,5.559,149.046
C00817=1200.782,-46.155,-41.090,179.770,5.558,149.046
C00818=1200.786,-46.405,-41.079,179.768,5.558,149.047
C00819=1200.792,-46.654,-41.066,179.765,5.557,149.048
C00820=1200.797,-46.904,-41.055,179.763,5.558,149.048
C00821=1200.802,-47.153,-41.042,179.760,5.557,149.049
C00822=1200.808,-47.403,-41.030,179.758,5.557,149.050
C00823=1200.812,-47.653,-41.019,179.756,5.557,149.050
C00824=1200.817,-47.902,-41.006,179.753,5.556,149.051
C00825=1200.823,-48.152,-40.994,179.751,5.556,149.052
C00826=1200.828,-48.402,-40.982,179.749,5.556,149.052
C00827=1200.833,-48.651,-40.970,179.746,5.556,149.053
C00828=1200.839,-48.922,-40.957,179.743,5.555,149.054
C00829=1200.845,-49.191,-40.944,179.741,5.555,149.054
C00830=1200.850,-49.462,-40.931,179.738,5.555,149.055
C00831=1200.856,-49.731,-40.919,179.736,5.555,149.056
C00832=1200.861,-49.981,-40.907,179.733,5.554,149.056
C00833=1200.866,-50.231,-40.896,179.730,5.554,149.057
C00834=1200.871,-50.480,-40.883,179.729,5.554,149.058
C00835=1200.876,-50.730,-40.871,179.726,5.553,149.058
C00836=1200.882,-50.980,-40.859,179.724,5.553,149.059
C00837=1200.887,-51.230,-40.848,179.721,5.553,149.060
C00838=1200.892,-51.479,-40.835,179.719,5.553,149.060
C00839=1200.897,-51.729,-40.823,179.716,5.552,149.061
C00840=1200.902,-51.979,-40.812,179.715,5.552,149.062
C00841=1200.907,-52.228,-40.800,179.712,5.552,149.062
C00842=1200.912,-52.478,-40.788,179.709,5.551,149.063
C00843=1200.918,-52.728,-40.776,179.707,5.552,149.064
C00844=1200.922,-52.977,-40.764,179.704,5.551,149.064
C00845=1200.928,-53.227,-40.753,179.702,5.551,149.065
C00846=1200.933,-53.477,-40.741,179.700,5.551,149.066
C00847=1200.938,-53.726,-40.729,179.698,5.550,149.066
C00848=1200.943,-53.976,-40.717,179.695,5.550,149.067
C00849=1200.949,-54.226,-40.705,179.693,5.550,149.068
C00850=1200.954,-54.475,-40.694,179.690,5.550,149.068
C00851=1200.959,-54.725,-40.682,179.688,5.549,149.069
C00852=1200.964,-54.975,-40.671,179.686,5.549,149.070
C00853=1200.969,-55.224,-40.658,179.683,5.549,149.070
C00854=1200.975,-55.474,-40.646,179.681,5.549,149.071
C00855=1200.979,-55.723,-40.635,179.678,5.549,149.072
C00856=1200.985,-55.973,-40.623,179.676,5.548,149.072
C00857=1200.990,-56.223,-40.611,179.674,5.548,149.073
C00858=1200.995,-56.473,-40.600,179.672,5.548,149.074
C00859=1201.000,-56.723,-40.588,179.669,5.548,149.074
C00860=1201.005,-56.972,-40.577,179.667,5.548,149.075
C00861=1201.011,-57.222,-40.565,179.664,5.547,149.076
C00862=1201.016,-57.471,-40.554,179.661,5.547,149.076
C00863=1201.021,-57.721,-40.542,179.660,5.547,149.077
C00864=1201.026,-57.971,-40.529,179.657,5.547,149.078
C00865=1201.031,-58.220,-40.518,179.655,5.546,149.078
C00866=1201.036,-58.470,-40.506,179.652,5.546,149.079
C00867=1201.041,-58.720,-40.495,179.650,5.546,149.080
C00868=1201.047,-58.969,-40.484,179.648,5.545,149.080
C00869=1201.052,-59.219,-40.472,179.646,5.546,149.081
C00870=1201.057,-59.469,-40.460,179.643,5.545,149.082
C00871=1201.062,-59.718,-40.449,179.640,5.545,149.082
C00872=1201.067,-59.968,-40.437,179.638,5.545,149.083
C00873=1201.073,-60.218,-40.425,179.635,5.545,149.084
C00874=1201.078,-60.467,-40.414,179.634,5.545,149.084
C00875=1201.083,-60.717,-40.402,179.631,5.544,149.085
C00876=1201.088,-60.967,-40.391,179.628,5.544,149.086
C00877=1201.094,-61.217,-40.379,179.626,5.544,149.086
C00878=1201.098,-61.466,-40.368,179.624,5.544,149.087
C00879=1201.104,-61.716,-40.356,179.622,5.543,149.088
C00880=1201.109,-61.966,-40.346,179.619,5.543,149.088
C00881=1201.115,-62.216,-40.334,179.617,5.543,149.089
C00882=1201.119,-62.465,-40.323,179.614,5.542,149.090
C00883=1201.125,-62.715,-40.311,179.612,5.543,149.090
C00884=1201.129,-62.965,-40.300,179.609,5.542,149.091
C00885=1201.135,-63.214,-40.289,179.608,5.542,149.092
C00886=1201.140,-63.464,-40.277,179.605,5.542,149.092
C00887=1201.145,-63.713,-40.265,179.602,5.541,149.093
C00888=1201.150,-63.963,-40.254,179.600,5.542,149.094
C00889=1201.156,-64.212,-40.243,179.598,5.541,149.094
C00890=1201.161,-64.463,-40.231,179.596,5.540,149.095
C00891=1201.166,-64.712,-40.220,179.593,5.541,149.096
C00892=1201.171,-64.962,-40.208,179.591,5.540,149.096
C00893=1201.176,-65.212,-40.197,179.589,5.541,149.097
C00894=1201.181,-65.461,-40.186,179.586,5.540,149.098
C00895=1201.187,-65.711,-40.174,179.584,5.539,149.098
C00896=1201.192,-65.960,-40.163,179.582,5.540,149.099
C00897=1201.197,-66.211,-40.152,179.579,5.539,149.100
C00898=1201.203,-66.460,-40.141,179.576,5.539,149.100
C00899=1201.208,-66.710,-40.129,179.574,5.539,149.101
C00900=1201.213,-66.959,-40.118,179.572,5.538,149.101
C00901=1201.217,-67.209,-40.106,179.570,5.539,149.102
C00902=1201.224,-67.459,-40.096,179.567,5.538,149.103
C00903=1201.228,-67.708,-40.084,179.565,5.538,149.104
C00904=1201.233,-67.958,-40.073,179.563,5.538,149.104
C00905=1201.239,-68.207,-40.061,179.560,5.537,149.105
C00906=1201.244,-68.458,-40.051,179.558,5.538,149.105
C00907=1201.250,-68.708,-40.039,179.556,5.537,149.106
C00908=1201.254,-68.957,-40.028,179.553,5.537,149.107
C00909=1201.260,-69.206,-40.017,179.551,5.537,149.108
C00910=1201.265,-69.457,-40.006,179.549,5.536,149.108
C00911=1201.270,-69.706,-39.994,179.546,5.536,149.109
C00912=1201.275,-69.955,-39.983,179.544,5.536,149.109
C00913=1201.281,-70.206,-39.972,179.541,5.536,149.110
C00914=1201.286,-70.455,-39.961,179.539,5.536,149.111
C00915=1201.291,-70.704,-39.950,179.537,5.536,149.111
C00916=1201.296,-70.954,-39.938,179.534,5.535,149.112
C00917=1201.301,-71.204,-39.928,179.532,5.535,149.113
C00918=1201.307,-71.453,-39.917,179.530,5.535,149.113
C00919=1201.312,-71.703,-39.905,179.528,5.535,149.114
C00920=1201.317,-71.954,-39.894,179.525,5.535,149.115
C00921=1201.322,-72.203,-39.883,179.523,5.534,149.115
C00922=1201.327,-72.453,-39.873,179.521,5.535,149.116
C00923=1201.333,-72.703,-39.861,179.518,5.534,149.117
C00924=1201.338,-72.952,-39.850,179.516,5.534,149.117
C00925=1201.343,-73.202,-39.839,179.514,5.534,149.118
C00926=1201.348,-73.451,-39.828,179.511,5.533,149.119
C00927=1201.354,-73.701,-39.816,179.509,5.534,149.119
C00928=1201.359,-73.951,-39.806,179.506,5.533,149.120
C00929=1201.364,-74.201,-39.795,179.504,5.534,149.121
C00930=1201.370,-74.450,-39.784,179.502,5.533,149.121
C00931=1201.375,-74.700,-39.773,179.499,5.532,149.122
C00932=1201.380,-74.971,-39.760,179.497,5.533,149.123
C00933=1201.386,-75.241,-39.749,179.495,5.532,149.123
C00934=1201.391,-75.512,-39.737,179.492,5.532,149.124
C00935=1201.398,-75.782,-39.725,179.490,5.532,149.125
C00936=1201.403,-76.033,-39.714,179.487,5.532,149.126
C00937=1201.407,-76.282,-39.703,179.484,5.531,149.126
C00938=1201.413,-76.532,-39.693,179.482,5.532,149.127
C00939=1201.418,-76.782,-39.681,179.480,5.531,149.127
C00940=1201.424,-77.031,-39.671,179.478,5.531,149.128
C00941=1201.429,-77.281,-39.659,179.475,5.531,149.129
C00942=1201.434,-77.531,-39.649,179.473,5.530,149.130
C00943=1201.439,-77.780,-39.638,179.471,5.531,149.130
C00944=1201.445,-78.031,-39.627,179.469,5.530,149.131
C00945=1201.450,-78.279,-39.616,179.466,5.530,149.131
C00946=1201.455,-78.530,-39.605,179.464,5.530,149.132
C00947=1201.460,-78.779,-39.594,179.462,5.530,149.133
C00948=1201.465,-79.029,-39.584,179.459,5.529,149.133
C00949=1201.470,-79.279,-39.573,179.457,5.529,149.134
C00950=1201.475,-79.528,-39.562,179.455,5.529,149.135
C00951=1201.481,-79.779,-39.551,179.452,5.529,149.135
C00952=1201.486,-80.028,-39.540,179.450,5.529,149.136
C00953=1201.491,-80.278,-39.530,179.448,5.528,149.137
C00954=1201.497,-80.527,-39.519,179.446,5.529,149.137
C00955=1201.502,-80.777,-39.508,179.443,5.528,149.138
C00956=1201.507,-81.027,-39.497,179.440,5.528,149.139
C00957=1201.512,-81.276,-39.487,179.439,5.528,149.139
C00958=1201.517,-81.526,-39.476,179.436,5.528,149.140
C00959=1201.522,-81.775,-39.465,179.434,5.528,149.141
C00960=1201.528,-82.026,-39.454,179.431,5.528,149.141
C00961=1201.534,-82.275,-39.444,179.429,5.528,149.142
C00962=1201.538,-82.525,-39.432,179.427,5.527,149.143
C00963=1201.544,-82.775,-39.422,179.424,5.527,149.143
C00964=1201.549,-83.025,-39.412,179.422,5.527,149.144
C00965=1201.554,-83.274,-39.401,179.420,5.527,149.145
C00966=1201.559,-83.524,-39.390,179.418,5.527,149.145
C00967=1201.565,-83.773,-39.380,179.415,5.526,149.146
C00968=1201.570,-84.023,-39.369,179.413,5.527,149.147
C00969=1201.575,-84.273,-39.358,179.411,5.526,149.147
C00970=1201.580,-84.523,-39.348,179.408,5.525,149.148
C00971=1201.585,-84.772,-39.337,179.406,5.526,149.149
C00972=1201.590,-85.022,-39.326,179.404,5.525,149.149
C00973=1201.596,-85.272,-39.316,179.402,5.526,149.150
C00974=1201.601,-85.522,-39.306,179.399,5.525,149.151
C00975=1201.606,-85.771,-39.295,179.397,5.525,149.151
C00976=1201.611,-86.021,-39.284,179.395,5.525,149.152
C00977=1201.617,-86.271,-39.274,179.392,5.524,149.153
C00978=1201.622,-86.521,-39.263,179.390,5.525,149.153
C00979=1201.627,-86.770,-39.252,179.388,5.524,149.154
C00980=1201.632,-87.020,-39.242,179.386,5.524,149.154
C00981=1201.638,-87.270,-39.232,179.383,5.524,149.155
C00982=1201.643,-87.520,-39.221,179.381,5.524,149.156
C00983=1201.648,-87.769,-39.210,179.379,5.523,149.156
C00984=1201.653,-88.019,-39.199,179.377,5.524,149.157
C00985=1201.659,-88.268,-39.189,179.374,5.523,149.158
C00986=1201.664,-88.519,-39.179,179.372,5.524,149.158
C00987=1201.669,-88.768,-39.168,179.370,5.523,149.159
C00988=1201.675,-89.017,-39.158,179.367,5.523,149.160
C00989=1201.680,-89.267,-39.147,179.365,5.523,149.160
C00990=1201.685,-89.517,-39.137,179.362,5.523,149.161
C00991=1201.690,-89.767,-39.126,179.361,5.523,149.162
C00992=1201.696,-90.017,-39.116,179.358,5.522,149.162
C00993=1201.701,-90.267,-39.105,179.356,5.522,149.163
C00994=1201.705,-90.516,-39.095,179.353,5.522,149.164
C00995=1201.711,-90.765,-39.085,179.352,5.522,149.164
C00996=1201.716,-91.015,-39.074,179.349,5.522,149.165
C00997=1201.722,-91.265,-39.064,179.346,5.521,149.166
C00998=1201.727,-91.515,-39.054,179.344,5.522,149.166
C00999=1201.732,-91.765,-39.043,179.342,5.521,149.167
C01000=1201.738,-92.014,-39.033,179.340,5.521,149.168
C01001=1201.743,-92.265,-39.023,179.337,5.521,149.168
C01002=1201.748,-92.514,-39.012,179.335,5.521,149.169
C01003=1201.753,-92.764,-39.002,179.333,5.520,149.169
C01004=1201.758,-93.013,-38.991,179.331,5.521,149.170
C01005=1201.763,-93.262,-38.981,179.328,5.520,149.171
C01006=1201.768,-93.513,-38.971,179.326,5.521,149.172
C01007=1201.774,-93.762,-38.960,179.324,5.520,149.172
C01008=1201.779,-94.013,-38.950,179.322,5.520,149.173
C01009=1201.785,-94.262,-38.940,179.319,5.520,149.173
C01010=1201.790,-94.512,-38.929,179.316,5.519,149.174
C01011=1201.795,-94.762,-38.919,179.315,5.519,149.175
C01012=1201.800,-95.011,-38.909,179.312,5.519,149.175
C01013=1201.806,-95.261,-38.899,179.310,5.519,149.176
C01014=1201.811,-95.511,-38.888,179.307,5.519,149.177
C01015=1201.816,-95.760,-38.878,179.306,5.519,149.177
C01016=1201.821,-96.010,-38.869,179.303,5.519,149.178
C01017=1201.826,-96.260,-38.858,179.301,5.519,149.179
C01018=1201.832,-96.509,-38.848,179.299,5.518,149.179
C01019=1201.837,-96.759,-38.838,179.297,5.519,149.180
C01020=1201.842,-97.009,-38.827,179.294,5.518,149.181
C01021=1201.848,-97.259,-38.817,179.292,5.518,149.181
C01022=1201.853,-97.508,-38.807,179.290,5.518,149.182
C01023=1201.858,-97.758,-38.797,179.288,5.518,149.183
C01024=1201.864,-98.008,-38.787,179.285,5.518,149.183
C01025=1201.869,-98.258,-38.777,179.283,5.518,149.184
C01026=1201.874,-98.508,-38.767,179.281,5.517,149.184
C01027=1201.879,-98.757,-38.757,179.278,5.517,149.185
C01028=1201.885,-99.007,-38.747,179.276,5.517,149.186
C01029=1201.890,-99.257,-38.736,179.274,5.516,149.186
C01030=1201.895,-99.506,-38.726,179.272,5.517,149.187
C01031=1201.900,-99.756,-38.716,179.269,5.516,149.188
C01032=1201.906,-100.006,-38.706,179.267,5.517,149.188
C01033=1201.911,-100.256,-38.695,179.265,5.516,149.189
C01034=1201.916,-100.506,-38.686,179.263,5.516,149.190
C01035=1201.922,-100.755,-38.676,179.260,5.516,149.190
C01036=1201.927,-101.026,-38.665,179.258,5.516,149.191
C01037=1201.933,-101.298,-38.654,179.255,5.516,149.192
C01038=1201.938,-101.569,-38.643,179.253,5.516,149.193
C01039=1201.945,-101.841,-38.632,179.251,5.516,149.193
C01040=1201.949,-102.091,-38.622,179.248,5.515,149.194
C01041=1201.955,-102.340,-38.612,179.246,5.515,149.194
C01042=1201.960,-102.590,-38.602,179.244,5.515,149.195
C01043=1201.965,-102.839,-38.592,179.242,5.515,149.196
C01044=1201.970,-103.090,-38.583,179.239,5.515,149.196
C01045=1201.976,-103.340,-38.572,179.237,5.515,149.197
C01046=1201.981,-103.589,-38.563,179.235,5.515,149.198
C01047=1201.986,-103.838,-38.553,179.233,5.515,149.198
C01048=1201.991,-104.089,-38.542,179.230,5.514,149.199
C01049=1201.997,-104.338,-38.533,179.228,5.515,149.200
C01050=1202.002,-104.588,-38.523,179.226,5.514,149.200
C01051=1202.007,-104.837,-38.513,179.224,5.514,149.201
C01052=1202.012,-105.087,-38.503,179.221,5.514,149.202
C01053=1202.018,-105.338,-38.493,179.220,5.514,149.202
C01054=1202.023,-105.587,-38.484,179.217,5.513,149.203
C01055=1202.028,-105.836,-38.473,179.215,5.514,149.204
C01056=1202.034,-106.087,-38.464,179.212,5.513,149.204
C01057=1202.039,-106.336,-38.454,179.210,5.513,149.205
C01058=1202.044,-106.586,-38.444,179.208,5.513,149.205
C01059=1202.049,-106.835,-38.434,179.205,5.513,149.206
C01060=1202.055,-107.085,-38.425,179.204,5.513,149.207
C01061=1202.061,-107.335,-38.414,179.201,5.512,149.207
C01062=1202.065,-107.585,-38.404,179.199,5.513,149.208
C01063=1202.071,-107.835,-38.395,179.197,5.512,149.209
C01064=1202.076,-108.084,-38.385,179.195,5.512,149.209
C01065=1202.081,-108.334,-38.375,179.192,5.512,149.210
C01066=1202.086,-108.584,-38.366,179.190,5.512,149.210
C01067=1202.091,-108.834,-38.356,179.188,5.511,149.211
C01068=1202.097,-109.083,-38.345,179.186,5.512,149.212
C01069=1202.102,-109.333,-38.336,179.183,5.511,149.213
C01070=1202.108,-109.583,-38.326,179.181,5.511,149.213
C01071=1202.113,-109.833,-38.317,179.179,5.511,149.214
C01072=1202.118,-110.082,-38.307,179.176,5.511,149.215
C01073=1202.123,-110.332,-38.297,179.174,5.511,149.215
C01074=1202.129,-110.582,-38.288,179.172,5.511,149.216
C01075=1202.133,-110.832,-38.278,179.170,5.511,149.216
C01076=1202.139,-111.082,-38.269,179.168,5.511,149.217
C01077=1202.144,-111.331,-38.259,179.166,5.511,149.218
C01078=1202.150,-111.581,-38.249,179.163,5.511,149.218
C01079=1202.154,-111.831,-38.239,179.162,5.511,149.219
C01080=1202.160,-112.081,-38.229,179.159,5.510,149.220
C01081=1202.165,-112.330,-38.220,179.157,5.511,149.220
C01082=1202.171,-112.580,-38.210,179.155,5.510,149.221
C01083=1202.176,-112.830,-38.201,179.153,5.510,149.221
C01084=1202.182,-113.079,-38.191,179.150,5.510,149.222
C01085=1202.187,-113.329,-38.182,179.148,5.510,149.223
C01086=1202.192,-113.579,-38.172,179.146,5.509,149.223
C01087=1202.197,-113.829,-38.163,179.143,5.510,149.224
C01088=1202.202,-114.079,-38.152,179.141,5.509,149.225
C01089=1202.208,-114.329,-38.144,179.139,5.509,149.225
C01090=1202.213,-114.578,-38.133,179.137,5.509,149.226
C01091=1202.218,-114.828,-38.124,179.135,5.509,149.226
C01092=1202.224,-115.078,-38.114,179.132,5.509,149.227
C01093=1202.229,-115.328,-38.105,179.130,5.509,149.228
C01094=1202.235,-115.577,-38.095,179.128,5.508,149.228
C01095=1202.240,-115.827,-38.086,179.126,5.509,149.229
C01096=1202.245,-116.076,-38.077,179.123,5.508,149.230
C01097=1202.251,-116.326,-38.067,179.122,5.508,149.230
C01098=1202.255,-116.576,-38.057,179.119,5.508,149.231
C01099=1202.261,-116.826,-38.048,179.117,5.508,149.232
C01100=1202.266,-117.076,-38.038,179.115,5.507,149.232
C01101=1202.271,-117.326,-38.029,179.113,5.508,149.233
C01102=1202.277,-117.576,-38.020,179.110,5.507,149.234
C01103=1202.282,-117.825,-38.010,179.108,5.507,149.234
C01104=1202.288,-118.075,-38.001,179.106,5.507,149.235
C01105=1202.292,-118.324,-37.991,179.103,5.507,149.236
C01106=1202.298,-118.574,-37.982,179.101,5.507,149.236
C01107=1202.303,-118.824,-37.973,179.099,5.507,149.237
C01108=1202.308,-119.074,-37.963,179.097,5.506,149.237
C01109=1202.313,-119.323,-37.954,179.095,5.507,149.238
C01110=1202.319,-119.574,-37.945,179.093,5.507,149.239
C01111=1202.324,-119.823,-37.935,179.091,5.506,149.239
C01112=1202.330,-120.073,-37.925,179.089,5.507,149.240
C01113=1202.335,-120.323,-37.917,179.086,5.506,149.241
C01114=1202.340,-120.572,-37.907,179.084,5.506,149.241
C01115=1202.346,-120.822,-37.897,179.082,5.506,149.242
C01116=1202.351,-121.072,-37.889,179.080,5.506,149.243
C01117=1202.356,-121.321,-37.879,179.077,5.505,149.243
C01118=1202.362,-121.571,-37.869,179.075,5.506,149.244
C01119=1202.367,-121.822,-37.860,179.073,5.505,149.244
C01120=1202.371,-122.071,-37.851,179.071,5.505,149.245
C01121=1202.377,-122.321,-37.842,179.068,5.505,149.246
C01122=1202.383,-122.571,-37.832,179.067,5.505,149.246
C01123=1202.387,-122.820,-37.823,179.064,5.505,149.247
C01124=1202.393,-123.070,-37.814,179.062,5.505,149.248
C01125=1202.398,-123.320,-37.804,179.060,5.504,149.248
C01126=1202.404,-123.570,-37.795,179.058,5.505,149.249
C01127=1202.409,-123.819,-37.786,179.056,5.505,149.249
C01128=1202.414,-124.069,-37.777,179.053,5.504,149.250
C01129=1202.420,-124.319,-37.768,179.051,5.505,149.251
C01130=1202.425,-124.569,-37.759,179.049,5.504,149.251
C01131=1202.430,-124.818,-37.749,179.047,5.504,149.252
C01132=1202.436,-125.068,-37.740,179.044,5.504,149.253
C01133=1202.441,-125.318,-37.731,179.043,5.504,149.253
C01134=1202.446,-125.568,-37.722,179.040,5.503,149.254
C01135=1202.452,-125.818,-37.713,179.038,5.503,149.254
C01136=1202.456,-126.067,-37.703,179.036,5.503,149.255
C01137=1202.462,-126.317,-37.694,179.034,5.503,149.256
C01138=1202.468,-126.567,-37.685,179.031,5.503,149.256
C01139=1202.473,-126.817,-37.676,179.029,5.503,149.257
C01140=1202.051,-126.827,-37.714,179.025,5.506,149.259
C01141=1202.046,-126.578,-37.724,179.027,5.506,149.258
C01142=1202.041,-126.328,-37.733,179.030,5.507,149.258
C01143=1202.036,-126.078,-37.741,179.032,5.506,149.257
C01144=1202.030,-125.828,-37.751,179.034,5.507,149.256
C01145=1202.024,-125.579,-37.760,179.036,5.507,149.256
C01146=1202.019,-125.329,-37.768,179.038,5.507,149.255
C01147=1202.014,-125.080,-37.778,179.040,5.507,149.254
C01148=1202.008,-124.830,-37.788,179.043,5.507,149.254
C01149=1202.003,-124.580,-37.796,179.045,5.507,149.253
C01150=1201.998,-124.330,-37.805,179.047,5.508,149.253
C01151=1201.993,-124.081,-37.815,179.049,5.507,149.252
C01152=1201.987,-123.831,-37.824,179.052,5.508,149.251
C01153=1201.982,-123.581,-37.833,179.054,5.508,149.251
C01154=1201.977,-123.331,-37.842,179.056,5.509,149.250
C01155=1201.972,-123.082,-37.852,179.058,5.508,149.249
C01156=1201.966,-122.831,-37.861,179.060,5.508,149.249
C01157=1201.961,-122.582,-37.870,179.062,5.509,149.248
C01158=1201.956,-122.332,-37.879,179.064,5.508,149.248
C01159=1201.950,-122.082,-37.889,179.067,5.509,149.247
C01160=1201.945,-121.832,-37.898,179.069,5.509,149.246
C01161=1201.940,-121.582,-37.907,179.071,5.509,149.246
C01162=1201.934,-121.333,-37.917,179.073,5.509,149.245
C01163=1201.929,-121.083,-37.926,179.076,5.509,149.244
C01164=1201.924,-120.833,-37.935,179.078,5.509,149.244
C01165=1201.919,-120.584,-37.945,179.080,5.510,149.243
C01166=1201.913,-120.334,-37.954,179.082,5.509,149.242
C01167=1201.908,-120.084,-37.963,179.085,5.510,149.242
C01168=1201.902,-119.834,-37.973,179.086,5.510,149.241
C01169=1201.897,-119.585,-37.982,179.089,5.510,149.241
C01170=1201.892,-119.335,-37.991,179.091,5.510,149.240
C01171=1201.887,-119.085,-38.002,179.093,5.511,149.239
C01172=1201.882,-118.835,-38.011,179.095,5.510,149.239
C01173=1201.877,-118.585,-38.020,179.097,5.510,149.238
C01174=1201.871,-118.335,-38.030,179.100,5.511,149.237
C01175=1201.866,-118.085,-38.039,179.102,5.510,149.237
C01176=1201.861,-117.836,-38.048,179.104,5.511,149.236
C01177=1201.855,-117.586,-38.058,179.106,5.510,149.236
C01178=1201.850,-117.336,-38.067,179.109,5.511,149.235
C01179=1201.844,-117.087,-38.077,179.110,5.511,149.234
C01180=1201.839,-116.837,-38.086,179.113,5.511,149.234
C01181=1201.834,-116.588,-38.095,179.115,5.511,149.233
C01182=1201.828,-116.337,-38.105,179.117,5.512,149.232
C01183=1201.823,-116.088,-38.114,179.119,5.511,149.232
C01184=1201.818,-115.838,-38.124,179.122,5.512,149.231
C01185=1201.813,-115.588,-38.133,179.124,5.512,149.230
C01186=1201.808,-115.338,-38.143,179.126,5.512,149.230
C01187=1201.802,-115.088,-38.152,179.128,5.512,149.229
C01188=1201.798,-114.839,-38.162,179.130,5.512,149.229
C01189=1201.792,-114.589,-38.171,179.133,5.512,149.228
C01190=1201.787,-114.339,-38.181,179.135,5.512,149.227
C01191=1201.781,-114.089,-38.191,179.137,5.512,149.227
C01192=1201.776,-113.840,-38.200,179.140,5.513,149.226
C01193=1201.770,-113.590,-38.210,179.142,5.512,149.225
C01194=1201.765,-113.341,-38.219,179.144,5.513,149.225
C01195=1201.759,-113.090,-38.229,179.146,5.513,149.224
C01196=1201.755,-112.841,-38.239,179.149,5.513,149.223
C01197=1201.749,-112.590,-38.248,179.150,5.513,149.223
C01198=1201.744,-112.341,-38.258,179.153,5.514,149.222
C01199=1201.738,-112.091,-38.267,179.155,5.513,149.221
C01200=1201.734,-111.842,-38.277,179.157,5.514,149.221
C01201=1201.728,-111.592,-38.287,179.159,5.514,149.220
C01202=1201.723,-111.342,-38.296,179.162,5.514,149.219
C01203=1201.717,-111.093,-38.306,179.163,5.514,149.219
C01204=1201.713,-110.842,-38.316,179.166,5.514,149.218
C01205=1201.707,-110.593,-38.326,179.168,5.514,149.218
C01206=1201.702,-110.343,-38.335,179.170,5.515,149.217
C01207=1201.696,-110.093,-38.345,179.173,5.514,149.216
C01208=1201.691,-109.844,-38.354,179.175,5.515,149.216
C01209=1201.685,-109.594,-38.364,179.177,5.515,149.215
C01210=1201.681,-109.344,-38.374,179.180,5.515,149.214
C01211=1201.675,-109.094,-38.383,179.182,5.515,149.214
C01212=1201.670,-108.845,-38.393,179.184,5.516,149.213
C01213=1201.665,-108.595,-38.403,179.186,5.515,149.213
C01214=1201.659,-108.345,-38.413,179.189,5.516,149.212
C01215=1201.654,-108.096,-38.422,179.190,5.516,149.211
C01216=1201.649,-107.845,-38.433,179.193,5.516,149.211
C01217=1201.644,-107.596,-38.442,179.195,5.516,149.210
C01218=1201.638,-107.346,-38.452,179.197,5.517,149.209
C01219=1201.633,-107.097,-38.462,179.199,5.516,149.209
C01220=1201.628,-106.847,-38.471,179.202,5.517,149.208
C01221=1201.623,-106.596,-38.482,179.203,5.517,149.208
C01222=1201.618,-106.347,-38.491,179.206,5.517,149.207
C01223=1201.612,-106.098,-38.502,179.208,5.517,149.206
C01224=1201.607,-105.848,-38.510,179.211,5.517,149.205
C01225=1201.601,-105.598,-38.521,179.212,5.517,149.205
C01226=1201.596,-105.348,-38.531,179.215,5.517,149.204
C01227=1201.591,-105.098,-38.540,179.217,5.517,149.203
C01228=1201.586,-104.849,-38.550,179.219,5.518,149.203
C01229=1201.580,-104.599,-38.561,179.222,5.517,149.202
C01230=1201.576,-104.349,-38.570,179.224,5.518,149.202
C01231=1201.570,-104.099,-38.580,179.226,5.518,149.201
C01232=1201.564,-103.849,-38.590,179.228,5.518,149.200
C01233=1201.559,-103.600,-38.600,179.231,5.518,149.200
C01234=1201.554,-103.350,-38.610,179.233,5.518,149.199
C01235=1201.549,-103.101,-38.620,179.235,5.518,149.198
C01236=1201.544,-102.851,-38.629,179.238,5.519,149.198
C01237=1201.538,-102.601,-38.640,179.240,5.518,149.197
C01238=1201.534,-102.351,-38.650,179.242,5.519,149.197
C01239=1201.528,-102.101,-38.660,179.244,5.519,149.196
C01240=1201.523,-101.852,-38.670,179.247,5.519,149.195
C01241=1201.517,-101.580,-38.680,179.249,5.519,149.194
C01242=1201.511,-101.308,-38.692,179.251,5.519,149.194
C01243=1201.505,-101.038,-38.702,179.254,5.519,149.193
C01244=1201.500,-100.766,-38.713,179.256,5.519,149.192
C01245=1201.494,-100.516,-38.723,179.258,5.520,149.192
C01246=1201.489,-100.266,-38.733,179.260,5.520,149.191
C01247=1201.484,-100.017,-38.744,179.263,5.520,149.190
C01248=1201.479,-99.767,-38.753,179.265,5.520,149.190
C01249=1201.474,-99.517,-38.764,179.267,5.520,149.189
C01250=1201.468,-99.268,-38.774,179.270,5.521,149.188
C01251=1201.463,-99.018,-38.784,179.272,5.520,149.188
C01252=1201.458,-98.769,-38.794,179.274,5.521,149.187
C01253=1201.452,-98.518,-38.804,179.276,5.521,149.187
C01254=1201.447,-98.268,-38.814,179.279,5.521,149.186
C01255=1201.442,-98.019,-38.824,179.281,5.521,149.185
C01256=1201.437,-97.769,-38.834,179.283,5.522,149.185
C01257=1201.431,-97.519,-38.844,179.285,5.521,149.184
C01258=1201.426,-97.270,-38.855,179.288,5.522,149.183
C01259=1201.421,-97.020,-38.865,179.290,5.522,149.183
C01260=1201.416,-96.770,-38.875,179.292,5.522,149.182
C01261=1201.410,-96.521,-38.885,179.294,5.522,149.181
C01262=1201.405,-96.271,-38.896,179.297,5.522,149.181
C01263=1201.400,-96.021,-38.906,179.299,5.522,149.180
C01264=1201.394,-95.771,-38.916,179.301,5.523,149.179
C01265=1201.390,-95.522,-38.926,179.303,5.522,149.179
C01266=1201.384,-95.272,-38.936,179.306,5.523,149.178
C01267=1201.379,-95.022,-38.946,179.308,5.523,149.177
C01268=1201.374,-94.772,-38.957,179.310,5.523,149.177
C01269=1201.368,-94.523,-38.967,179.313,5.523,149.176
C01270=1201.362,-94.273,-38.977,179.315,5.523,149.176
C01271=1201.358,-94.023,-38.987,179.317,5.524,149.175
C01272=1201.353,-93.774,-38.997,179.319,5.523,149.174
C01273=1201.348,-93.523,-39.008,179.322,5.524,149.173
C01274=1201.342,-93.274,-39.018,179.324,5.524,149.173
C01275=1201.336,-93.024,-39.028,179.326,5.524,149.172
C01276=1201.331,-92.774,-39.039,179.328,5.524,149.172
C01277=1201.326,-92.525,-39.049,179.331,5.524,149.171
C01278=1201.321,-92.275,-39.059,179.333,5.524,149.170
C01279=1201.316,-92.025,-39.069,179.335,5.525,149.170
C01280=1201.311,-91.776,-39.080,179.338,5.525,149.169
C01281=1201.306,-91.526,-39.091,179.340,5.525,149.168
C01282=1201.300,-91.276,-39.101,179.342,5.526,149.168
C01283=1201.295,-91.026,-39.112,179.344,5.525,149.167
C01284=1201.289,-90.777,-39.122,179.347,5.526,149.166
C01285=1201.284,-90.527,-39.132,179.349,5.525,149.166
C01286=1201.279,-90.277,-39.143,179.351,5.526,149.165
C01287=1201.273,-90.027,-39.153,179.353,5.526,149.164
C01288=1201.268,-89.777,-39.164,179.356,5.526,149.164
C01289=1201.264,-89.528,-39.174,179.358,5.526,149.163
C01290=1201.258,-89.279,-39.184,179.360,5.526,149.162
C01291=1201.253,-89.029,-39.195,179.363,5.527,149.162
C01292=1201.248,-88.779,-39.205,179.365,5.527,149.161
C01293=1201.243,-88.529,-39.215,179.367,5.527,149.161
C01294=1201.237,-88.280,-39.226,179.369,5.527,149.160
C01295=1201.232,-88.030,-39.237,179.372,5.527,149.159
C01296=1201.227,-87.780,-39.247,179.374,5.527,149.158
C01297=1201.222,-87.530,-39.258,179.377,5.527,149.158
C01298=1201.216,-87.280,-39.268,179.378,5.527,149.157
C01299=1201.211,-87.031,-39.279,179.381,5.528,149.157
C01300=1201.206,-86.781,-39.289,179.384,5.528,149.156
C01301=1201.200,-86.532,-39.300,179.386,5.528,149.155
C01302=1201.195,-86.281,-39.310,179.388,5.529,149.155
C01303=1201.190,-86.032,-39.321,179.390,5.528,149.154
C01304=1201.185,-85.782,-39.332,179.393,5.529,149.153
C01305=1201.179,-85.533,-39.342,179.395,5.528,149.153
C01306=1201.174,-85.282,-39.352,179.397,5.529,149.152
C01307=1201.169,-85.033,-39.363,179.399,5.529,149.151
C01308=1201.164,-84.783,-39.374,179.402,5.529,149.151
C01309=1201.158,-84.534,-39.384,179.405,5.530,149.150
C01310=1201.153,-84.283,-39.395,179.406,5.530,149.149
C01311=1201.148,-84.034,-39.406,179.409,5.530,149.149
C01312=1201.143,-83.784,-39.416,179.411,5.530,149.148
C01313=1201.138,-83.535,-39.426,179.414,5.530,149.147
C01314=1201.133,-83.285,-39.438,179.415,5.530,149.147
C01315=1201.127,-83.036,-39.448,179.418,5.531,149.146
C01316=1201.122,-82.785,-39.459,179.421,5.531,149.145
C01317=1201.117,-82.536,-39.469,179.423,5.531,149.145
C01318=1201.112,-82.286,-39.480,179.425,5.531,149.144
C01319=1201.106,-82.036,-39.491,179.427,5.531,149.143
C01320=1201.101,-81.787,-39.502,179.430,5.531,149.143
C01321=1201.096,-81.536,-39.513,179.432,5.531,149.142
C01322=1201.091,-81.287,-39.524,179.434,5.532,149.141
C01323=1201.086,-81.037,-39.534,179.437,5.532,149.141
C01324=1201.080,-80.788,-39.544,179.439,5.532,149.140
C01325=1201.075,-80.538,-39.556,179.441,5.532,149.139
C01326=1201.070,-80.288,-39.566,179.443,5.532,149.139
C01327=1201.065,-80.039,-39.577,179.446,5.533,149.138
C01328=1201.059,-79.789,-39.587,179.448,5.532,149.138
C01329=1201.054,-79.539,-39.599,179.450,5.533,149.137
C01330=1201.049,-79.289,-39.610,179.453,5.533,149.136
C01331=1201.043,-79.040,-39.620,179.455,5.533,149.135
C01332=1201.039,-78.790,-39.631,179.457,5.534,149.135
C01333=1201.033,-78.540,-39.642,179.459,5.533,149.134
C01334=1201.028,-78.291,-39.653,179.462,5.534,149.134
C01335=1201.023,-78.041,-39.663,179.464,5.533,149.133
C01336=1201.017,-77.791,-39.675,179.466,5.534,149.132
C01337=1201.012,-77.541,-39.686,179.469,5.535,149.132
C01338=1201.007,-77.292,-39.696,179.471,5.534,149.131
C01339=1201.002,-77.042,-39.707,179.474,5.535,149.130
C01340=1200.997,-76.793,-39.718,179.476,5.534,149.130
C01341=1200.991,-76.542,-39.729,179.478,5.535,149.129
C01342=1200.986,-76.293,-39.740,179.481,5.536,149.128
C01343=1200.981,-76.043,-39.751,179.483,5.535,149.128
C01344=1200.976,-75.794,-39.762,179.485,5.536,149.127
C01345=1200.970,-75.523,-39.774,179.487,5.535,149.126
C01346=1200.964,-75.252,-39.785,179.490,5.536,149.125
C01347=1200.959,-74.981,-39.797,179.493,5.536,149.125
C01348=1200.953,-74.711,-39.809,179.496,5.537,149.124
C01349=1200.948,-74.461,-39.820,179.498,5.536,149.123
C01350=1200.942,-74.211,-39.831,179.500,5.537,149.123
C01351=1200.937,-73.962,-39.842,179.502,5.537,149.122
C01352=1200.932,-73.712,-39.854,179.505,5.537,149.121
C01353=1200.927,-73.463,-39.864,179.507,5.538,149.121
C01354=1200.921,-73.213,-39.876,179.509,5.537,149.120
C01355=1200.916,-72.962,-39.886,179.511,5.538,149.120
C01356=1200.911,-72.713,-39.897,179.514,5.538,149.119
C01357=1200.906,-72.463,-39.909,179.516,5.538,149.118
C01358=1200.901,-72.213,-39.920,179.519,5.538,149.117
C01359=1200.895,-71.964,-39.931,179.520,5.538,149.117
C01360=1200.891,-71.715,-39.942,179.523,5.539,149.116
C01361=1200.885,-71.464,-39.953,179.525,5.539,149.116
C01362=1200.880,-71.215,-39.964,179.528,5.539,149.115
C01363=1200.875,-70.966,-39.975,179.531,5.539,149.114
C01364=1200.869,-70.715,-39.986,179.532,5.539,149.114
C01365=1200.864,-70.466,-39.997,179.535,5.540,149.113
C01366=1200.859,-70.216,-40.009,179.537,5.539,149.112
C01367=1200.854,-69.966,-40.020,179.540,5.540,149.112
C01368=1200.848,-69.717,-40.031,179.542,5.540,149.111
C01369=1200.844,-69.467,-40.042,179.544,5.540,149.110
C01370=1200.838,-69.217,-40.053,179.547,5.541,149.110
C01371=1200.833,-68.967,-40.064,179.549,5.541,149.109
C01372=1200.828,-68.718,-40.075,179.551,5.541,149.108
C01373=1200.822,-68.468,-40.087,179.554,5.541,149.108
C01374=1200.817,-68.218,-40.098,179.556,5.541,149.107
C01375=1200.812,-67.969,-40.109,179.558,5.542,149.106
C01376=1200.807,-67.719,-40.121,179.561,5.542,149.106
C01377=1200.802,-67.470,-40.132,179.563,5.542,149.105
C01378=1200.796,-67.219,-40.143,179.566,5.542,149.104
C01379=1200.791,-66.970,-40.154,179.567,5.542,149.104
C01380=1200.786,-66.721,-40.165,179.570,5.543,149.103
C01381=1200.781,-66.471,-40.177,179.573,5.543,149.102
C01382=1200.776,-66.222,-40.188,179.575,5.543,149.102
C01383=1200.770,-65.971,-40.199,179.577,5.543,149.101
C01384=1200.765,-65.721,-40.211,179.580,5.544,149.100
C01385=1200.760,-65.472,-40.222,179.582,5.544,149.100
C01386=1200.754,-65.223,-40.233,179.584,5.544,149.099
C01387=1200.750,-64.973,-40.245,179.586,5.544,149.098
C01388=1200.744,-64.723,-40.257,179.589,5.544,149.098
C01389=1200.739,-64.473,-40.267,179.591,5.545,149.097
C01390=1200.735,-64.223,-40.278,179.593,5.545,149.096
C01391=1200.729,-63.974,-40.290,179.596,5.545,149.096
C01392=1200.724,-63.724,-40.301,179.599,5.546,149.095
C01393=1200.718,-63.474,-40.313,179.601,5.545,149.094
C01394=1200.714,-63.225,-40.324,179.603,5.546,149.094
C01395=1200.708,-62.976,-40.336,179.605,5.546,149.093
C01396=1200.703,-62.726,-40.347,179.608,5.546,149.092
C01397=1200.698,-62.476,-40.359,179.610,5.547,149.092
C01398=1200.693,-62.226,-40.370,179.612,5.546,149.091
C01399=1200.687,-61.976,-40.382,179.615,5.547,149.090
C01400=1200.682,-61.727,-40.392,179.617,5.547,149.090
C01401=1200.676,-61.477,-40.404,179.619,5.547,149.089
C01402=1200.672,-61.227,-40.416,179.622,5.548,149.088
C01403=1200.666,-60.977,-40.428,179.624,5.547,149.088
C01404=1200.662,-60.728,-40.439,179.627,5.548,149.087
C01405=1200.656,-60.478,-40.451,179.629,5.548,149.087
C01406=1200.651,-60.229,-40.462,179.631,5.548,149.086
C01407=1200.646,-59.979,-40.474,179.634,5.548,149.085
C01408=1200.641,-59.729,-40.485,179.636,5.549,149.084
C01409=1200.635,-59.479,-40.497,179.638,5.549,149.084
C01410=1200.631,-59.230,-40.508,179.641,5.549,149.083
C01411=1200.625,-58.980,-40.520,179.643,5.550,149.083
C01412=1200.620,-58.731,-40.531,179.645,5.549,149.082
C01413=1200.615,-58.481,-40.543,179.648,5.550,149.081
C01414=1200.609,-58.231,-40.555,179.651,5.550,149.080
C01415=1200.604,-57.981,-40.566,179.653,5.550,149.080
C01416=1200.599,-57.731,-40.578,179.655,5.551,149.079
C01417=1200.594,-57.482,-40.589,179.658,5.551,149.079
C01418=1200.589,-57.232,-40.601,179.660,5.551,149.078
C01419=1200.584,-56.983,-40.612,179.662,5.551,149.077
C01420=1200.578,-56.734,-40.624,179.664,5.551,149.076
C01421=1200.573,-56.484,-40.636,179.667,5.552,149.076
C01422=1200.568,-56.234,-40.648,179.669,5.552,149.075
C01423=1200.563,-55.984,-40.659,179.671,5.552,149.075
C01424=1200.558,-55.735,-40.671,179.674,5.552,149.074
C01425=1200.553,-55.485,-40.683,179.677,5.553,149.073
C01426=1200.547,-55.235,-40.695,179.679,5.552,149.072
C01427=1200.543,-54.985,-40.706,179.681,5.553,149.072
C01428=1200.537,-54.735,-40.718,179.684,5.554,149.071
C01429=1200.532,-54.487,-40.729,179.686,5.553,149.071
C01430=1200.527,-54.237,-40.741,179.688,5.554,149.070
C01431=1200.521,-53.987,-40.753,179.691,5.554,149.069
C01432=1200.517,-53.737,-40.764,179.693,5.554,149.068
C01433=1200.511,-53.487,-40.776,179.695,5.555,149.068
C01434=1200.506,-53.237,-40.788,179.698,5.555,149.067
C01435=1200.501,-52.988,-40.800,179.700,5.555,149.067
C01436=1200.496,-52.738,-40.812,179.703,5.555,149.066
C01437=1200.491,-52.489,-40.824,179.705,5.556,149.065
C01438=1200.486,-52.239,-40.835,179.707,5.556,149.065
C01439=1200.480,-51.989,-40.847,179.710,5.556,149.064
C01440=1200.475,-51.740,-40.860,179.712,5.557,149.063
C01441=1200.470,-51.490,-40.872,179.714,5.556,149.063
C01442=1200.465,-51.240,-40.883,179.717,5.557,149.062
C01443=1200.460,-50.990,-40.895,179.720,5.557,149.061
C01444=1200.454,-50.742,-40.907,179.721,5.557,149.061
C01445=1200.449,-50.492,-40.918,179.724,5.558,149.060
C01446=1200.444,-50.242,-40.930,179.727,5.558,149.059
C01447=1200.439,-49.992,-40.942,179.729,5.558,149.059
C01448=1200.433,-49.743,-40.955,179.731,5.558,149.058
C01449=1200.428,-49.472,-40.968,179.734,5.559,149.057
C01450=1200.423,-49.202,-40.981,179.737,5.559,149.056
C01451=1200.417,-48.932,-40.993,179.739,5.560,149.056
C01452=1200.412,-48.662,-41.006,179.741,5.559,149.055
C01453=1200.406,-48.412,-41.018,179.744,5.560,149.054
C01454=1200.401,-48.163,-41.031,179.747,5.560,149.054
C01455=1200.396,-47.913,-41.042,179.748,5.560,149.053
C01456=1200.391,-47.663,-41.054,179.751,5.561,149.052
C01457=1200.386,-47.414,-41.066,179.754,5.561,149.052
C01458=1200.380,-47.164,-41.078,179.756,5.561,149.051
C01459=1200.375,-46.914,-41.090,179.758,5.561,149.050
C01460=1200.371,-46.665,-41.102,179.761,5.562,149.050
C01461=1200.365,-46.415,-41.114,179.763,5.562,149.049
C01462=1200.360,-46.165,-41.126,179.765,5.562,149.048
C01463=1200.355,-45.916,-41.139,179.768,5.563,149.048
C01464=1200.349,-45.666,-41.151,179.771,5.563,149.047
C01465=1200.345,-45.417,-41.163,179.773,5.563,149.046
C01466=1200.339,-45.167,-41.174,179.775,5.563,149.046
C01467=1200.334,-44.917,-41.186,179.778,5.564,149.045
C01468=1200.329,-44.668,-41.199,179.780,5.564,149.045
C01469=1200.323,-44.418,-41.211,179.782,5.564,149.044
C01470=1200.318,-44.168,-41.223,179.785,5.564,149.043
C01471=1200.313,-43.918,-41.235,179.787,5.564,149.042
C01472=1200.308,-43.669,-41.247,179.790,5.565,149.042
C01473=1200.303,-43.420,-41.259,179.792,5.565,149.041
C01474=1200.298,-43.170,-41.272,179.795,5.566,149.041
C01475=1200.293,-42.920,-41.284,179.797,5.566,149.040
C01476=1200.288,-42.670,-41.297,179.799,5.566,149.039
C01477=1200.282,-42.420,-41.308,179.802,5.566,149.038
C01478=1200.277,-42.171,-41.321,179.804,5.566,149.038
C01479=1200.272,-41.921,-41.333,179.806,5.567,149.037
C01480=1200.267,-41.672,-41.346,179.809,5.567,149.037
C01481=1200.261,-41.422,-41.357,179.811,5.567,149.036
C01482=1200.257,-41.173,-41.369,179.814,5.568,149.035
C01483=1200.252,-40.923,-41.381,179.816,5.568,149.034
C01484=1200.246,-40.674,-41.394,179.819,5.568,149.034
C01485=1200.241,-40.424,-41.406,179.821,5.568,149.033
C01486=1200.236,-40.174,-41.419,179.823,5.569,149.033
C01487=1200.231,-39.924,-41.431,179.826,5.569,149.032
C01488=1200.226,-39.674,-41.443,179.828,5.569,149.031
C01489=1200.221,-39.425,-41.456,179.831,5.569,149.030
C01490=1200.215,-39.175,-41.468,179.833,5.570,149.030
C01491=1200.210,-38.926,-41.480,179.836,5.571,149.029
C01492=1200.205,-38.676,-41.492,179.838,5.570,149.029
C01493=1200.200,-38.427,-41.505,179.840,5.571,149.028
C01494=1200.195,-38.177,-41.517,179.843,5.571,149.027
C01495=1200.190,-37.927,-41.530,179.845,5.571,149.026
C01496=1200.185,-37.677,-41.542,179.848,5.571,149.026
C01497=1200.179,-37.428,-41.555,179.850,5.572,149.025
C01498=1200.174,-37.178,-41.567,179.853,5.573,149.025
C01499=1200.169,-36.929,-41.579,179.855,5.572,149.024
C01500=1200.164,-36.679,-41.592,179.857,5.573,149.023
C01501=1200.158,-36.429,-41.604,179.860,5.573,149.023
C01502=1200.154,-36.179,-41.617,179.863,5.574,149.022
C01503=1200.149,-35.930,-41.629,179.864,5.574,149.021
C01504=1200.143,-35.680,-41.641,179.867,5.574,149.021
C01505=1200.138,-35.431,-41.654,179.870,5.575,149.020
C01506=1200.133,-35.182,-41.667,179.872,5.574,149.019
C01507=1200.128,-34.931,-41.679,179.874,5.575,149.019
C01508=1200.123,-34.682,-41.691,179.877,5.575,149.018
C01509=1200.118,-34.432,-41.704,179.879,5.576,149.017
C01510=1200.112,-34.183,-41.717,179.881,5.576,149.017
C01511=1200.107,-33.933,-41.729,179.884,5.576,149.016
C01512=1200.102,-33.683,-41.742,179.887,5.577,149.015
C01513=1200.097,-33.433,-41.755,179.889,5.577,149.015
C01514=1200.092,-33.184,-41.767,179.891,5.577,149.014
C01515=1200.087,-32.935,-41.780,179.893,5.578,149.013
C01516=1200.081,-32.685,-41.792,179.896,5.578,149.013
C01517=1200.076,-32.435,-41.804,179.899,5.579,149.012
C01518=1200.072,-32.185,-41.817,179.901,5.578,149.011
C01519=1200.067,-31.936,-41.830,179.903,5.579,149.011
C01520=1200.061,-31.686,-41.843,179.906,5.579,149.010
C01521=1200.055,-31.437,-41.855,179.908,5.580,149.009
C01522=1200.051,-31.187,-41.868,179.910,5.580,149.009
C01523=1200.046,-30.937,-41.881,179.913,5.580,149.008
C01524=1200.040,-30.688,-41.893,179.916,5.581,149.007
C01525=1200.035,-30.439,-41.906,179.918,5.580,149.007
C01526=1200.031,-30.189,-41.919,179.920,5.581,149.006
C01527=1200.025,-29.939,-41.932,179.923,5.581,149.005
C01528=1200.020,-29.689,-41.944,179.925,5.582,149.005
C01529=1200.014,-29.440,-41.956,179.928,5.583,149.004
C01530=1200.010,-29.190,-41.969,179.930,5.582,149.003
C01531=1200.005,-28.940,-41.982,179.933,5.583,149.003
C01532=1199.999,-28.691,-41.995,179.935,5.583,149.002
C01533=1199.994,-28.441,-42.008,179.938,5.584,149.001
C01534=1199.989,-28.191,-42.021,179.940,5.584,149.001
C01535=1199.984,-27.942,-42.033,179.942,5.584,149.000
C01536=1199.979,-27.693,-42.046,179.945,5.585,148.999
C01537=1199.974,-27.442,-42.059,179.948,5.585,148.999
C01538=1199.969,-27.193,-42.072,179.950,5.585,148.998
C01539=1199.964,-26.944,-42.085,179.952,5.585,148.997
C01540=1199.959,-26.694,-42.098,179.955,5.586,148.997
C01541=1199.954,-26.444,-42.110,179.957,5.587,148.996
C01542=1199.948,-26.195,-42.123,179.959,5.586,148.996
C01543=1199.943,-25.945,-42.136,179.962,5.587,148.995
C01544=1199.938,-25.695,-42.149,179.965,5.587,148.994
C01545=1199.933,-25.446,-42.162,179.967,5.588,148.993
C01546=1199.927,-25.197,-42.175,179.969,5.588,148.993
C01547=1199.923,-24.947,-42.188,179.971,5.588,148.992
C01548=1199.918,-24.697,-42.200,179.974,5.589,148.992
C01549=1199.912,-24.448,-42.214,179.977,5.589,148.991
C01550=1199.907,-24.198,-42.227,179.979,5.590,148.990
C01551=1199.902,-23.948,-42.239,179.982,5.589,148.989
C01552=1199.897,-23.699,-42.252,179.984,5.590,148.989
C01553=1199.891,-23.429,-42.266,179.987,5.590,148.988
C01554=1199.886,-23.159,-42.280,179.990,5.591,148.987
C01555=1199.881,-22.889,-42.294,179.992,5.591,148.987
C01556=1199.875,-22.620,-42.309,179.995,5.592,148.986
C01557=1199.870,-22.370,-42.322,179.998,5.592,148.985
C01558=1199.865,-22.121,-42.334,179.999,5.592,148.985
C01559=1199.859,-21.871,-42.347,-179.998,5.593,148.984
C01560=1199.855,-21.621,-42.360,-179.996,5.593,148.983
C01561=1199.849,-21.372,-42.373,-179.993,5.594,148.983
C01562=1199.844,-21.122,-42.386,-179.991,5.593,148.982
C01563=1199.839,-20.873,-42.400,-179.988,5.594,148.981
C01564=1199.834,-20.624,-42.412,-179.986,5.595,148.981
C01565=1199.829,-20.373,-42.426,-179.983,5.595,148.980
C01566=1199.824,-20.124,-42.439,-179.981,5.595,148.979
C01567=1199.818,-19.874,-42.452,-179.979,5.595,148.979
C01568=1199.813,-19.624,-42.465,-179.976,5.596,148.978
C01569=1199.809,-19.376,-42.478,-179.973,5.596,148.977
C01570=1199.803,-19.125,-42.492,-179.971,5.597,148.977
C01571=1199.798,-18.876,-42.504,-179.968,5.597,148.976
C01572=1199.792,-18.626,-42.517,-179.966,5.597,148.976
C01573=1199.788,-18.376,-42.530,-179.964,5.598,148.975
C01574=1199.783,-18.128,-42.544,-179.961,5.598,148.974
C01575=1199.778,-17.877,-42.557,-179.958,5.598,148.973
C01576=1199.773,-17.628,-42.570,-179.956,5.599,148.973
C01577=1199.767,-17.378,-42.583,-179.954,5.599,148.972
C01578=1199.763,-17.129,-42.597,-179.952,5.599,148.972
C01579=1199.757,-16.879,-42.610,-179.949,5.600,148.971
C01580=1199.752,-16.629,-42.623,-179.946,5.600,148.970
C01581=1199.747,-16.380,-42.637,-179.944,5.601,148.970
C01582=1199.742,-16.130,-42.650,-179.942,5.601,148.969
C01583=1199.737,-15.881,-42.662,-179.939,5.601,148.968
C01584=1199.732,-15.631,-42.677,-179.937,5.602,148.968
C01585=1199.727,-15.382,-42.689,-179.934,5.602,148.967
C01586=1199.722,-15.132,-42.703,-179.931,5.603,148.966
C01587=1199.717,-14.883,-42.716,-179.929,5.603,148.966
C01588=1199.712,-14.633,-42.730,-179.927,5.603,148.965
C01589=1199.706,-14.383,-42.742,-179.924,5.604,148.964
C01590=1199.701,-14.134,-42.756,-179.922,5.604,148.964
C01591=1199.696,-13.884,-42.769,-179.919,5.605,148.963
C01592=1199.691,-13.635,-42.782,-179.916,5.605,148.962
C01593=1199.686,-13.385,-42.796,-179.914,5.605,148.962
C01594=1199.680,-13.136,-42.809,-179.912,5.606,148.961
C01595=1199.675,-12.885,-42.823,-179.910,5.606,148.961
C01596=1199.670,-12.637,-42.836,-179.907,5.607,148.960
C01597=1199.665,-12.386,-42.850,-179.904,5.607,148.959
C01598=1199.660,-12.138,-42.863,-179.902,5.608,148.958
C01599=1199.655,-11.887,-42.877,-179.900,5.607,148.958
C01600=1199.651,-11.638,-42.890,-179.897,5.608,148.957
C01601=1199.645,-11.388,-42.903,-179.895,5.609,148.957
C01602=1199.641,-11.139,-42.917,-179.892,5.609,148.956
C01603=1199.635,-10.889,-42.930,-179.889,5.610,148.955
C01604=1199.630,-10.639,-42.944,-179.887,5.610,148.955
C01605=1199.625,-10.390,-42.957,-179.885,5.610,148.954
C01606=1199.620,-10.140,-42.971,-179.882,5.611,148.953
C01607=1199.615,-9.891,-42.984,-179.880,5.611,148.953
C01608=1199.609,-9.641,-42.998,-179.877,5.612,148.952
C01609=1199.604,-9.392,-43.012,-179.875,5.612,148.951
C01610=1199.599,-9.142,-43.025,-179.872,5.613,148.951
C01611=1199.594,-8.892,-43.039,-179.870,5.612,148.950
C01612=1199.589,-8.643,-43.053,-179.868,5.613,148.949
C01613=1199.584,-8.393,-43.066,-179.865,5.614,148.949
C01614=1199.579,-8.144,-43.080,-179.862,5.614,148.948
C01615=1199.574,-7.894,-43.093,-179.860,5.615,148.947
C01616=1199.569,-7.645,-43.106,-179.857,5.615,148.947
C01617=1199.563,-7.395,-43.120,-179.855,5.615,148.946
C01618=1199.559,-7.145,-43.134,-179.853,5.616,148.946
C01619=1199.554,-6.896,-43.148,-179.850,5.616,148.945
C01620=1199.548,-6.646,-43.161,-179.847,5.617,148.944
C01621=1199.544,-6.397,-43.174,-179.845,5.617,148.943
C01622=1199.538,-6.147,-43.188,-179.842,5.618,148.943
C01623=1199.533,-5.897,-43.202,-179.839,5.618,148.942
C01624=1199.528,-5.648,-43.216,-179.838,5.618,148.942
C01625=1199.523,-5.398,-43.229,-179.835,5.619,148.941
C01626=1199.518,-5.149,-43.243,-179.833,5.619,148.940
C01627=1199.513,-4.900,-43.257,-179.830,5.620,148.940
C01628=1199.508,-4.649,-43.270,-179.827,5.620,148.939
C01629=1199.503,-4.400,-43.284,-179.825,5.621,148.938
C01630=1199.498,-4.151,-43.299,-179.822,5.621,148.938
C01631=1199.492,-3.900,-43.312,-179.820,5.621,148.937
C01632=1199.488,-3.652,-43.325,-179.818,5.622,148.936
C01633=1199.483,-3.402,-43.340,-179.815,5.622,148.936
C01634=1199.477,-3.152,-43.353,-179.812,5.623,148.935
C01635=1199.472,-2.903,-43.367,-179.810,5.623,148.934
C01636=1199.468,-2.653,-43.381,-179.808,5.624,148.934
C01637=1199.462,-2.404,-43.394,-179.805,5.624,148.933
C01638=1199.457,-2.154,-43.408,-179.803,5.624,148.932
C01639=1199.452,-1.904,-43.423,-179.800,5.625,148.932
C01640=1199.447,-1.656,-43.436,-179.798,5.625,148.931
C01641=1199.442,-1.406,-43.450,-179.795,5.626,148.931
C01642=1199.437,-1.155,-43.464,-179.793,5.626,148.930
C01643=1199.431,-0.906,-43.478,-179.790,5.627,148.929
C01644=1199.426,-0.657,-43.492,-179.787,5.627,148.928
C01645=1199.421,-0.407,-43.506,-179.785,5.628,148.928
C01646=1199.417,-0.157,-43.519,-179.783,5.628,148.927
C01647=1199.411,0.092,-43.533,-179.781,5.628,148.927
C01648=1199.406,0.342,-43.547,-179.778,5.629,148.926
C01649=1199.401,0.591,-43.562,-179.775,5.629,148.925
C01650=1199.396,0.840,-43.576,-179.773,5.630,148.925
C01651=1199.391,1.090,-43.590,-179.770,5.630,148.924
C01652=1199.386,1.340,-43.603,-179.768,5.631,148.923
C01653=1199.381,1.589,-43.617,-179.765,5.632,148.923
C01654=1199.376,1.839,-43.631,-179.762,5.632,148.922
C01655=1199.371,2.089,-43.645,-179.760,5.632,148.921
C01656=1199.366,2.338,-43.660,-179.758,5.632,148.921
C01657=1199.360,2.607,-43.674,-179.755,5.633,148.920
C01658=1199.355,2.876,-43.690,-179.752,5.633,148.919
C01659=1199.349,3.145,-43.705,-179.750,5.634,148.919
C01660=1199.344,3.415,-43.720,-179.747,5.634,148.918
C01661=1199.339,3.664,-43.734,-179.744,5.635,148.917
C01662=1199.333,3.913,-43.748,-179.742,5.636,148.917
C01663=1199.328,4.163,-43.762,-179.740,5.636,148.916
C01664=1199.324,4.413,-43.777,-179.737,5.637,148.915
C01665=1199.319,4.662,-43.791,-179.734,5.637,148.915
C01666=1199.313,4.911,-43.805,-179.732,5.638,148.914
C01667=1199.308,5.161,-43.819,-179.729,5.638,148.913
C01668=1199.304,5.411,-43.833,-179.727,5.639,148.913
C01669=1199.299,5.660,-43.847,-179.724,5.640,148.912
C01670=1199.294,5.910,-43.861,-179.722,5.639,148.912
C01671=1199.288,6.159,-43.875,-179.719,5.640,148.911
C01672=1199.283,6.409,-43.890,-179.717,5.640,148.910
C01673=1199.278,6.658,-43.904,-179.715,5.641,148.910
C01674=1199.274,6.908,-43.918,-179.712,5.642,148.909
C01675=1199.269,7.158,-43.932,-179.709,5.642,148.908
C01676=1199.263,7.407,-43.946,-179.707,5.643,148.908
C01677=1199.258,7.657,-43.961,-179.704,5.643,148.907
C01678=1199.253,7.906,-43.975,-179.702,5.644,148.906
C01679=1199.248,8.156,-43.989,-179.699,5.645,148.906
C01680=1199.243,8.406,-44.003,-179.697,5.645,148.905
C01681=1199.238,8.655,-44.017,-179.694,5.646,148.904
C01682=1199.233,8.904,-44.032,-179.692,5.645,148.904
C01683=1199.228,9.153,-44.047,-179.689,5.646,148.903
C01684=1199.223,9.403,-44.061,-179.687,5.647,148.903
C01685=1199.217,9.653,-44.076,-179.684,5.647,148.902
C01686=1199.212,9.903,-44.090,-179.682,5.648,148.901
C01687=1199.207,10.152,-44.104,-179.679,5.648,148.901
C01688=1199.202,10.402,-44.118,-179.676,5.649,148.900
C01689=1199.197,10.651,-44.132,-179.674,5.649,148.899
C01690=1199.192,10.900,-44.147,-179.672,5.650,148.899
C01691=1199.187,11.150,-44.162,-179.669,5.650,148.898
C01692=1199.182,11.400,-44.176,-179.666,5.651,148.897
C01693=1199.177,11.650,-44.190,-179.664,5.651,148.897
C01694=1199.172,11.899,-44.205,-179.662,5.652,148.896
C01695=1199.167,12.148,-44.218,-179.659,5.653,148.896
C01696=1199.162,12.397,-44.233,-179.657,5.653,148.895
C01697=1199.157,12.647,-44.248,-179.654,5.653,148.894
C01698=1199.152,12.897,-44.263,-179.652,5.654,148.893
C01699=1199.147,13.147,-44.277,-179.649,5.654,148.893
C01700=1199.142,13.396,-44.292,-179.647,5.655,148.892
C01701=1199.137,13.646,-44.306,-179.644,5.655,148.892
C01702=1199.132,13.895,-44.320,-179.641,5.656,148.891
C01703=1199.127,14.145,-44.335,-179.639,5.656,148.890
C01704=1199.121,14.394,-44.350,-179.637,5.657,148.890
C01705=1199.116,14.643,-44.364,-179.634,5.658,148.889
C01706=1199.111,14.893,-44.378,-179.631,5.658,148.888
C01707=1199.107,15.142,-44.393,-179.629,5.659,148.888
C01708=1199.102,15.392,-44.408,-179.626,5.659,148.887
C01709=1199.097,15.642,-44.422,-179.624,5.660,148.887
C01710=1199.091,15.891,-44.438,-179.621,5.661,148.886
C01711=1199.086,16.141,-44.452,-179.619,5.661,148.885
C01712=1199.081,16.391,-44.466,-179.616,5.662,148.885
C01713=1199.077,16.640,-44.481,-179.613,5.662,148.884
C01714=1199.072,16.889,-44.495,-179.611,5.663,148.883
C01715=1199.066,17.139,-44.510,-179.609,5.663,148.883
C01716=1199.061,17.388,-44.525,-179.606,5.663,148.882
C01717=1199.057,17.638,-44.540,-179.604,5.664,148.881
C01718=1199.052,17.888,-44.554,-179.601,5.664,148.881
C01719=1199.046,18.137,-44.569,-179.599,5.665,148.880
C01720=1199.041,18.387,-44.584,-179.596,5.666,148.880
C01721=1199.037,18.636,-44.599,-179.594,5.666,148.879
C01722=1199.032,18.886,-44.613,-179.591,5.667,148.878
C01723=1199.026,19.135,-44.629,-179.589,5.668,148.878
C01724=1199.021,19.384,-44.642,-179.586,5.668,148.877
C01725=1199.016,19.634,-44.657,-179.584,5.669,148.876
C01726=1199.010,19.883,-44.672,-179.581,5.669,148.876
C01727=1199.005,20.133,-44.687,-179.578,5.670,148.875
C01728=1199.001,20.382,-44.702,-179.576,5.670,148.875
C01729=1198.996,20.632,-44.716,-179.573,5.671,148.874
C01730=1198.991,20.882,-44.732,-179.571,5.671,148.873
C01731=1198.986,21.132,-44.746,-179.568,5.672,148.873
C01732=1198.981,21.381,-44.761,-179.565,5.673,148.872
C01733=1198.976,21.631,-44.776,-179.563,5.673,148.871
C01734=1198.971,21.880,-44.791,-179.561,5.674,148.871
C01735=1198.966,22.130,-44.805,-179.558,5.674,148.870
C01736=1198.961,22.379,-44.821,-179.555,5.675,148.869
C01737=1198.956,22.628,-44.836,-179.553,5.676,148.869
C01738=1198.951,22.878,-44.850,-179.551,5.676,148.868
C01739=1198.946,23.127,-44.866,-179.548,5.677,148.868
C01740=1198.941,23.377,-44.880,-179.545,5.677,148.867
C01741=1198.935,23.626,-44.896,-179.543,5.678,148.866
C01742=1198.930,23.876,-44.910,-179.540,5.679,148.866
C01743=1198.926,24.125,-44.925,-179.538,5.679,148.865
C01744=1198.920,24.374,-44.940,-179.535,5.680,148.864
C01745=1198.915,24.624,-44.955,-179.533,5.680,148.864
C01746=1198.910,24.874,-44.970,-179.530,5.681,148.863
C01747=1198.905,25.123,-44.985,-179.528,5.682,148.863
C01748=1198.900,25.372,-45.000,-179.525,5.682,148.862
C01749=1198.895,25.622,-45.015,-179.522,5.683,148.861
C01750=1198.891,25.872,-45.030,-179.520,5.683,148.861
C01751=1198.885,26.122,-45.045,-179.518,5.684,148.860
C01752=1198.881,26.371,-45.060,-179.515,5.685,148.859
C01753=1198.875,26.621,-45.075,-179.512,5.685,148.859
C01754=1198.870,26.870,-45.090,-179.510,5.686,148.858
C01755=1198.866,27.119,-45.105,-179.508,5.686,148.858
C01756=1198.860,27.368,-45.121,-179.505,5.687,148.857
C01757=1198.855,27.618,-45.135,-179.502,5.687,148.856
C01758=1198.850,27.867,-45.151,-179.500,5.688,148.856
C01759=1198.846,28.117,-45.166,-179.497,5.689,148.855
C01760=1198.841,28.367,-45.182,-179.495,5.689,148.854
C01761=1198.835,28.635,-45.197,-179.492,5.690,148.854
C01762=1198.830,28.905,-45.214,-179.490,5.690,148.853
C01763=1198.824,29.173,-45.231,-179.487,5.691,148.852
C01764=1198.819,29.442,-45.246,-179.484,5.692,148.852
C01765=1198.813,29.691,-45.262,-179.481,5.693,148.851
C01766=1198.809,29.940,-45.277,-179.478,5.693,148.850
C01767=1198.803,30.190,-45.293,-179.476,5.694,148.850
C01768=1198.798,30.439,-45.307,-179.474,5.695,148.849
C01769=1198.794,30.689,-45.323,-179.471,5.695,148.849
C01770=1198.789,30.939,-45.338,-179.468,5.696,148.848
C01771=1198.784,31.188,-45.353,-179.466,5.696,148.847
C01772=1198.779,31.437,-45.368,-179.463,5.697,148.847
C01773=1198.774,31.686,-45.384,-179.461,5.698,148.846
C01774=1198.768,31.936,-45.399,-179.458,5.698,148.845
C01775=1198.764,32.186,-45.414,-179.456,5.699,148.845
C01776=1198.758,32.436,-45.430,-179.453,5.700,148.844
C01777=1198.754,32.685,-45.445,-179.451,5.700,148.844
C01778=1198.748,32.934,-45.460,-179.448,5.701,148.843
C01779=1198.744,33.183,-45.475,-179.445,5.701,148.842
C01780=1198.739,33.433,-45.491,-179.443,5.702,148.842
C01781=1198.734,33.683,-45.507,-179.441,5.703,148.841
C01782=1198.729,33.932,-45.522,-179.438,5.703,148.840
C01783=1198.724,34.181,-45.537,-179.435,5.704,148.840
C01784=1198.719,34.431,-45.553,-179.433,5.704,148.839
C01785=1198.714,34.681,-45.568,-179.431,5.705,148.839
C01786=1198.708,34.930,-45.583,-179.428,5.705,148.838
C01787=1198.703,35.180,-45.599,-179.425,5.706,148.837
C01788=1198.698,35.429,-45.614,-179.423,5.708,148.837
C01789=1198.694,35.679,-45.630,-179.420,5.708,148.836
C01790=1198.689,35.928,-45.645,-179.417,5.709,148.836
C01791=1198.684,36.178,-45.660,-179.415,5.709,148.835
C01792=1198.678,36.427,-45.676,-179.412,5.710,148.834
C01793=1198.673,36.677,-45.692,-179.410,5.711,148.834
C01794=1198.669,36.926,-45.708,-179.407,5.711,148.833
C01795=1198.664,37.175,-45.723,-179.405,5.712,148.832
C01796=1198.658,37.424,-45.739,-179.402,5.713,148.832
C01797=1198.654,37.674,-45.754,-179.400,5.713,148.831
C01798=1198.649,37.924,-45.770,-179.397,5.714,148.831
C01799=1198.643,38.173,-45.785,-179.394,5.714,148.830
C01800=1198.639,38.423,-45.801,-179.392,5.715,148.829
C01801=1198.634,38.672,-45.816,-179.390,5.716,148.829
C01802=1198.629,38.922,-45.832,-179.387,5.716,148.828
C01803=1198.623,39.171,-45.847,-179.384,5.717,148.827
C01804=1198.618,39.421,-45.863,-179.382,5.718,148.827
C01805=1198.614,39.670,-45.878,-179.379,5.719,148.826
C01806=1198.609,39.919,-45.895,-179.376,5.719,148.826
C01807=1198.604,40.169,-45.911,-179.374,5.720,148.825
C01808=1198.599,40.418,-45.926,-179.372,5.721,148.825
C01809=1198.594,40.668,-45.941,-179.369,5.721,148.824
C01810=1198.589,40.918,-45.957,-179.366,5.722,148.823
C01811=1198.584,41.167,-45.973,-179.364,5.723,148.823
C01812=1198.579,41.416,-45.989,-179.361,5.723,148.822
C01813=1198.574,41.666,-46.005,-179.359,5.724,148.821
C01814=1198.569,41.915,-46.020,-179.356,5.724,148.821
C01815=1198.564,42.164,-46.036,-179.354,5.725,148.820
C01816=1198.559,42.415,-46.052,-179.351,5.726,148.820
C01817=1198.554,42.663,-46.068,-179.348,5.727,148.819
C01818=1198.549,42.913,-46.083,-179.346,5.728,148.818
C01819=1198.544,43.163,-46.099,-179.343,5.729,148.818
C01820=1198.539,43.412,-46.114,-179.341,5.729,148.817
C01821=1198.534,43.661,-46.131,-179.338,5.730,148.816
C01822=1198.529,43.911,-46.147,-179.336,5.730,148.816
C01823=1198.524,44.160,-46.162,-179.333,5.731,148.815
C01824=1198.519,44.410,-46.179,-179.331,5.732,148.815
C01825=1198.514,44.659,-46.195,-179.328,5.732,148.814
C01826=1198.509,44.908,-46.210,-179.326,5.733,148.814
C01827=1198.504,45.159,-46.226,-179.323,5.734,148.813
C01828=1198.500,45.407,-46.242,-179.320,5.735,148.812
C01829=1198.494,45.656,-46.257,-179.318,5.736,148.812
C01830=1198.489,45.907,-46.273,-179.315,5.736,148.811
C01831=1198.484,46.155,-46.290,-179.313,5.737,148.810
C01832=1198.479,46.405,-46.306,-179.310,5.737,148.810
C01833=1198.474,46.654,-46.322,-179.308,5.738,148.809
C01834=1198.470,46.904,-46.338,-179.305,5.739,148.809
